	(*TODO: Implement temperature Errors specific to current Cryo MODE (COLD, WARM etc): LOWLOW, LOW, OKAY, HIGH, HIGHHIGH*)
	{attribute 'OPC.UA.DA' := '0'}
	in_lrLowWarning:		LREAL;
	{attribute 'OPC.UA.DA' := '0'}
	in_lrLowLowAlarm:		LREAL;
	{attribute 'OPC.UA.DA' := '0'}
	in_lrHighWarning:		LREAL;
	{attribute 'OPC.UA.DA' := '0'}
	in_HighHighAlarm:		LREAL;
	
END_VAR
VAR
	{attribute 'OPC.UA.DA' := '0'}
	i_fValue	AT%I*:	REAL;    // lower precision, used e.g. by LS240
	{attribute 'OPC.UA.DA' := '0'}
	i_lrValue	AT%I*:  LREAL;   // higher precision, used by other sources
	{attribute 'OPC.UA.DA' := '0'}
    i_bValid    AT%I*:	BOOL;    // valid status, used e.g. by ramp and voters
		
    {attribute 'OPC.UA.DA' := '0'}
	RefStatBase:    REFERENCE TO T_METIS_SENSOR_BASE_STATUS;
	
	{attribute 'OPC.UA.DA' := '0'}
	bRampTimerStarted:	BOOL := FALSE;
	{attribute 'OPC.UA.DA' := '0'}
	rampTimer:	TON;		// Timer for calculating ramp
	
END_VAR

// Set references
RefStat	REF= RefStatBase;


// Get the raw reading and the status of the input channel
M_ReadSensor();

// Calculate value and validity
M_SetStatus();

// Calculate Temperature change ramp
M_GetRamp();

METHOD M_GetRamp
VAR_INPUT
END_VAR
VAR_INST
	{attribute 'OPC.UA.DA' := '0'}
	lrRampStartValueSi: LREAL;	// SI value at start of ramp timer [K]
END_VAR
VAR
	nRampPeriodSec:		UDINT;	// Ramp measurement period [sec].
END_VAR
IF NOT bRampTimerStarted THEN
	bRampTimerStarted	:= TRUE;
	lrRampStartValueSi	:= RefStatBase.lrBaseValue;
	rampTimer(IN:=FALSE);
END_IF

// Execute timer.
// Ramp measurement period should be > 0
nRampPeriodSec	:= in_nRampPeriodSec;
IF nRampPeriodSec = 0 THEN
	nRampPeriodSec	:= 60;
END_IF
rampTimer(IN:=TRUE,PT:=UDINT_TO_TIME(nRampPeriodSec)*1000);

// Calculate ramp at time expiry
IF rampTimer.Q THEN
	// Calculate the temperature ramp per minute
    RefStatBase.lrBaseRamp := (RefStatBase.lrBaseValue - lrRampStartValueSi) * 60.0 / nRampPeriodSec;

	// Current temperature is the starting value of the ramp
	lrRampStartValueSi := RefStatBase.lrBaseValue;

	// Restart the timer
	rampTimer(IN:=FALSE);
END_IF
END_METHOD

// Get input channel status and the raw reading
METHOD M_ReadSensor
VAR_INPUT
END_VAR
VAR_INST
    {attribute 'OPC.UA.DA' := '0'}
    lrPreviousBaseValue : LREAL;
    
    {attribute 'OPC.UA.DA' := '0'}
    _changingValueTimeout : TON;
END_VAR
// Get the base value
CASE in_eSource OF 
    E_METIS_SENSOR_SOURCE.LS240:
        RefStatBase.lrBaseValue := REAL_TO_LREAL(i_fValue) * in_lrScale + in_lrOffset;
    E_METIS_SENSOR_SOURCE.LS336,
    E_METIS_SENSOR_SOURCE.VOTER,
    E_METIS_SENSOR_SOURCE.RAMP,
    E_METIS_SENSOR_SOURCE.DEW_POINT_CALC:
        RefStatBase.lrBaseValue := i_lrValue * in_lrScale + in_lrOffset;
    E_METIS_SENSOR_SOURCE.EL32XX:
        SUPER^.M_ReadSensor();
        RefStatBase.lrBaseValue := INT_TO_LREAL(i_nValue) * in_lrScale + in_lrOffset;
    ELSE
        RefStatBase.lrBaseValue := i_lrValue * in_lrScale + in_lrOffset;
END_CASE

// check if the value is changing
IF RefStatBase.lrBaseValue <> lrPreviousBaseValue THEN
    _changingValueTimeout(IN := FALSE);
    lrPreviousBaseValue := RefStatBase.lrBaseValue;
ELSE
    IF in_eSource = E_METIS_SENSOR_SOURCE.LS240 THEN
        _changingValueTimeout(IN := TRUE, PT := T#20s);
    ELSE
        _changingValueTimeout(IN := TRUE, PT := T#60s);
	END_IF
END_IF

// use the changing value to set the status for sources that don't have a better
// status indication
CASE in_eSource OF 
    E_METIS_SENSOR_SOURCE.EL32XX:
        ; // already set by SUPER^.M_ReadSensor()
    E_METIS_SENSOR_SOURCE.LS240:
        RefStat.bInputUnder	    := FALSE;
        RefStat.bInputOver	    := FALSE;
        RefStat.bInputToggle    := FALSE;
        RefStat.bInputError	    := FALSE;
        RefStat.bInputValid	    := NOT _changingValueTimeout.Q;
        RefStat.bInputActive    := RefStat.bInputValid;
    ELSE
        RefStat.bInputUnder	    := FALSE;
        RefStat.bInputOver	    := FALSE;
        RefStat.bInputToggle    := FALSE;
        RefStat.bInputError	    := NOT i_bValid;
        RefStat.bInputValid     := i_bValid AND (NOT _changingValueTimeout.Q);
        RefStat.bInputActive    := i_bValid AND (NOT _changingValueTimeout.Q);
END_CASE
END_METHOD

METHOD M_SetStatus
VAR_INPUT
END_VAR
// TODO USER: Implement the method.

// copy some input values to the stat object
RefStatBase.eType    := in_eType;
RefStatBase.eSource  := in_eSource;
RefStatBase.sName    := in_sName;

// Update value depending on the sensor type.
// So far, only PT100 supported.

IF RefStat.bInputActive THEN
    
    CASE in_eSource OF
        E_METIS_SENSOR_SOURCE.LS240:
            M_SetStatus_LS240();
        E_METIS_SENSOR_SOURCE.EL32XX:
			RefStat.bError			:= RefStat.bInputError OR RefStat.bInputOver OR RefStat.bInputUnder;
        	RefStat.bValid 	        := NOT RefStat.bError;
        	RefStatBase.bWarning    := FALSE; 
			IF RefStat.bInputOver THEN
        		RefStatBase.sErrorText  := 'OVERRANGE';
			ELSIF RefStat.bInputUnder THEN
        		RefStatBase.sErrorText  := 'UNDERRANGE';
			ELSIF RefStat.bInputError THEN
        		RefStatBase.sErrorText  := 'INPUT ERROR';
			ELSIF RefStat.bError THEN
        		RefStatBase.sErrorText  := 'ERROR';
			ELSE
        		RefStatBase.sErrorText  := 'VALID READING';
			END_IF
    ELSE
        RefStat.bValid 	        := TRUE; 
        RefStat.bError 	        := FALSE;
        RefStatBase.bWarning    := FALSE; 
        RefStatBase.sErrorText  := 'VALID READING';
    END_CASE
ELSE	
	RefStat.bValid	        := FALSE;
	RefStat.bError	        := TRUE;
	RefStatBase.bWarning    := FALSE;
    RefStatBase.sErrorText  := 'INACTIVE';
END_IF
END_METHOD

// Calculate pressure based on the status in input value
METHOD M_SetStatus_LS240
VAR_INPUT
END_VAR
VAR
	lr_MaxRamp:		LREAL := in_lrFaultRamp + 10.0;

	lr_T_LowError:		LREAL := 25.0;
	lr_T_LowWarning:	LREAL := 30.0;
	lr_T_HighWarning:	LREAL := 345.0;
	lr_T_HighError:		LREAL := 346.0;  
END_VAR

IF RefStatBase.lrBaseValue > lr_T_LowWarning AND RefStatBase.lrBaseValue < lr_T_HighWarning AND
    ABS(RefStatBase.lrBaseRamp) < in_lrFaultRamp THEN
    
    RefStat.bValid          := TRUE; 
    RefStatBase.bWarning     := FALSE; 
    RefStat.bError          := FALSE;
    RefStatBase.sErrorText   := 'WITHIN RANGE';
    
ELSIF (RefStatBase.lrBaseValue < lr_T_LowWarning AND RefStatBase.lrBaseValue > lr_T_LowError) OR
        (RefStatBase.lrBaseValue > lr_T_HighWarning AND RefStatBase.lrBaseValue < lr_T_HighError) OR
        ABS(RefStatBase.lrBaseRamp) > in_lrFaultRamp AND ABS(RefStatBase.lrBaseRamp) < lr_MaxRamp THEN

    RefStat.bValid          := TRUE;
    RefStatBase.bWarning     := TRUE;  
    RefStat.bError          := FALSE;
    RefStatBase.sErrorText   := 'WARNING LIMITS EXCEEDED';
    
ELSIF RefStatBase.lrBaseValue < lr_T_LowError OR RefStatBase.lrBaseValue > lr_T_HighError OR
    ABS(RefStatBase.lrBaseRamp) > lr_MaxRamp THEN
    
    RefStat.bValid          := FALSE;
    RefStatBase.bWarning     := FALSE;	   
    RefStat.bError          := TRUE;
    RefStatBase.sErrorText   := 'ERROR LIMITS EXCEEDED';
   
END_IF
END_METHOD

END_FUNCTION_BLOCK

// POUs/Devices/Temp_Sensor/FB_SIM_TEMP_SENSOR_DT670
FUNCTION_BLOCK FB_SIM_TEMP_SENSOR_DT670
VAR_INPUT
	
	//in_lrTempK:		LREAL	:= 100.0;	// Target Temperature [K]
	in_Temp_Sensor_DT670:		FB_METIS_TEMP_SENSOR_DT670;	
	
END_VAR
VAR_OUTPUT
END_VAR
VAR
	sName											: STRING;	

	(* input *)
	bEnable											: BOOL		:= TRUE;
	fStart											: LREAL 	:= 100;
	fTarget											: LREAL		:= 150;
	
	bInit											: BOOL 		:= TRUE; (* To initialize the required ramp*)
	
	(* Ramp *)
	RampUp_Rate										: LREAL		:= 8;	(* in units per Minute *) 
	RampDown_Rate									: LREAL		:= 8;	(* in units per Minute *)
	
	(* function block *)
	fbCTRL_RAMP_GENERATOR							: FB_CTRL_RAMP_GENERATOR;
	stCTRL_RAMP_GENERATOR_PARAMS					: ST_CTRL_RAMP_GENERATOR_PARAMS;	
	
	q_bToggle	AT%Q*:	BOOL	:= FALSE;	// Simulated status
	q_fValue	AT%Q*:	REAL;			// Simulated value [bit]
	
	fOut				: LREAL;		
    bValueReached		: BOOL;
    bError				: BOOL;
    eErrorId			: E_CTRL_ERRORCODES;
	bConfigured			: BOOL;
	
////////////////////////////////////////////////////	
	
	{attribute 'OPC.UA.DA' := '0'}
	toggleTimer:	TON;		// Timer for PDO (alive) toggle
	{attribute 'OPC.UA.DA' := '0'}
	rampTimer:		TON;		// Timer for temperature ramp

	{attribute 'OPC.UA.DA' := '0'}
	nPeriod:		UDINT	:= 10000;	// RAMP/SINE Command period, default 10000ms = 10s
	
	lrTemp_SetPoint:			LREAL;
	
	
END_VAR

// Configuration 

sName := in_Temp_Sensor_DT670.in_sName;

IF bInit THEN
	M_Configure();
END_IF

stCTRL_RAMP_GENERATOR_PARAMS.fVeloPos			:= 0.01666 * RampUp_Rate; (* 1/60 to convert into units per second *)
stCTRL_RAMP_GENERATOR_PARAMS.fVeloNeg			:= 0.01666 * RampDown_Rate; (* 1/60 to convert into units per second *)

//ctrl.fTarget := in_fRampSetPoint;

// Execute Controller
M_ExecuteController();


// lrTempK
q_fValue	:= LREAL_TO_REAL(fOut);

//
// Simulate terminal alive toggle every 160ms.
//
IF NOT bEnable THEN
	bEnable	:= TRUE;
	toggleTimer(IN:=FALSE);
END_IF
toggleTimer(IN:=TRUE,PT:=T#160MS);

q_bToggle	:= toggleTimer.Q;
IF toggleTimer.Q THEN
	q_bToggle	:= toggleTimer.Q;
	toggleTimer(IN:=FALSE);
END_IF

METHOD M_Configure : BOOL
VAR_INPUT
END_VAR


(* init parameter struct *)
	stCTRL_RAMP_GENERATOR_PARAMS.tTaskCycleTime		:= T#10MS;
	stCTRL_RAMP_GENERATOR_PARAMS.tCtrlCycleTime		:= T#10MS;
	stCTRL_RAMP_GENERATOR_PARAMS.fVeloPos			:= 0.01666 * RampUp_Rate; (* 1/60 to convert into units per second *)
	stCTRL_RAMP_GENERATOR_PARAMS.fVeloNeg			:= 0.01666 * RampDown_Rate; (* 1/60 to convert into units per second *)

	(* reset the init flag *)
	bInit							:= FALSE;
END_METHOD

METHOD M_ExecuteController : BOOL
VAR_INPUT
END_VAR
(* call function block *)
fbCTRL_RAMP_GENERATOR(				bEnable					:= bEnable,
									fStart					:= fStart,
									fTarget					:= fTarget,
									stParams				:= stCTRL_RAMP_GENERATOR_PARAMS,
									fOut					=> fOut,
									bValueReached			=> bValueReached,
									bError					=> bError,
									eErrorId				=> eErrorId);
END_METHOD

END_FUNCTION_BLOCK

// POUs/Devices/Temp_Sensor/FB_METIS_TEMP_SENSOR_DT670
FUNCTION_BLOCK FB_METIS_TEMP_SENSOR_DT670
VAR_INPUT
	{attribute 'OPC.UA.DA' := '0'}
	in_sName:				STRING;
	{attribute 'OPC.UA.DA' := '0'}
	in_nLSType:				E_METIS_LAKE_SHORE_TYPE	:= E_METIS_LAKE_SHORE_TYPE.LS240;
	{attribute 'OPC.UA.DA' := '0'}
	in_nRampPeriodSec:		UDINT := 60;		// Ramp measurement period [sec]. Default 60 sec.
	{attribute 'OPC.UA.DA' := '0'}
	in_lrFaultRamp:			LREAL := 10;		// Ramp > in_nFaultRamp OR Ramp < -in_nFaultRamp(deg/min) indicate DT670 sensor fault.	

	(*TODO: Implement temperature Errors specific to current Cryo MODE (COLD, WARM etc): LOWLOW, LOW, OKAY, HIGH, HIGHHIGH*)
	{attribute 'OPC.UA.DA' := '0'}
	in_lrLowWarning:		LREAL;
	{attribute 'OPC.UA.DA' := '0'}
	in_lrLowLowAlarm:		LREAL;
	{attribute 'OPC.UA.DA' := '0'}
	in_lrHighWarning:		LREAL;
	{attribute 'OPC.UA.DA' := '0'}
	in_HighHighAlarm:		LREAL;
	
	in_nCryoMode:			INT; // COLD, COOL_DOWN, WARM_UP, WARM

END_VAR
VAR
//	{attribute 'OPC.UA.DA' := '0'}
//	i_nStatus	AT %I*: UINT;
	{attribute 'OPC.UA.DA' := '0'}
	i_fValue	AT%I*:	REAL;   // lower precision, used by LS240
	{attribute 'OPC.UA.DA' := '0'}
	i_lrValue	AT%I*:  LREAL;   // higher precision, used by other sources
	{attribute 'OPC.UA.DA' := '0'}
	i_bToggle	AT%I*:	BOOL;
	
	{attribute 'OPC.UA.DA' := '0'}
	bStarted:		BOOL := FALSE;
	{attribute 'OPC.UA.DA' := '0'}
	toggleTimer:	TON;		// Timer for PDO (alive) toggle
	{attribute 'OPC.UA.DA' := '0'}
	toggleTrig:		R_TRIG;		// PDO (alive) toggle detection
	
	RefStat: 	REFERENCE TO T_METIS_DT670_TEMP_SENSOR_STATUS;
	
	{attribute 'OPC.UA.DA' := '0'}
	stat:	T_METIS_DT670_TEMP_SENSOR_STATUS;	// Complete status

	{attribute 'OPC.UA.DA' := '0'}
	bRampTimerStarted:	BOOL := FALSE;
	{attribute 'OPC.UA.DA' := '0'}
	rampTimer:	TON;		// Timer for calculating ramp
	
END_VAR

// Set references
RefStat	REF=stat;


// Get the raw reading and the status of the input channel
M_ReadSensor();

// Calculate value and validity
M_SetStatus();

// Calculate Temperature change ramp
M_GetRamp();

METHOD M_GetRamp
VAR_INPUT
END_VAR
VAR_INST
	{attribute 'OPC.UA.DA' := '0'}
	lrRampStartTempK:	LREAL;	// Temperature at start of ramp timer [K]
END_VAR
VAR
	nRampPeriodSec:		UDINT;	// Ramp measurement period [sec].
END_VAR
IF NOT bRampTimerStarted THEN
	bRampTimerStarted	:= TRUE;
	lrRampStartTempK	:= stat.lrTempK;
	rampTimer(IN:=FALSE);
END_IF

// Execute timer.
// Ramp measurement period should be > 0
nRampPeriodSec	:= in_nRampPeriodSec;
IF nRampPeriodSec = 0 THEN
	nRampPeriodSec	:= 60;
END_IF
rampTimer(IN:=TRUE,PT:=UDINT_TO_TIME(nRampPeriodSec)*1000);

// Calculate ramp at time expiry
IF rampTimer.Q THEN
	// Calculate the temperature ramp per minute
//	IF stat.bValid THEN
		stat.lrRamp	:= (stat.lrTempK - lrRampStartTempK) * 60.0 / nRampPeriodSec;
//	ELSE
//		stat.lrRamp	:= 0.0;
//	END_IF

	// Current temperature is the starting value of the ramp
	lrRampStartTempK	:= stat.lrTempK;

	// Restart the timer
	rampTimer(IN:=FALSE);
END_IF
END_METHOD

// Get input channel status and the raw reading
METHOD M_ReadSensor
VAR_INPUT
END_VAR
VAR_INST
    fPreviousValue : REAL;
END_VAR
// Get input channel status
//RefStat.bInputUnder	:= (i_nStatus AND 2#0000_0000_0000_0001) <> 0;
//RefStat.bInputOver	:= (i_nStatus AND 2#0000_0000_0000_0010) <> 0;
//RefStat.bInputError	:= (i_nStatus AND 2#0000_0000_0100_0000) <> 0;
//RefStat.bInputToggle:= (i_nStatus AND 2#1000_0000_0000_0000) <> 0;
//RefStat.bInputValid	:= (i_nStatus AND 2#0100_0000_0000_0000)  = 0;	// 0 -> PDO OK

// Get the raw reading
CASE in_nLSType OF 
    E_METIS_LAKE_SHORE_TYPE.LS240:
        RefStat.lrRawValue	:= REAL_TO_LREAL(i_fValue);
    E_METIS_LAKE_SHORE_TYPE.LS336,
    E_METIS_LAKE_SHORE_TYPE.VOTER,
    E_METIS_LAKE_SHORE_TYPE.RAMP:
        RefStat.lrRawValue	:= i_lrValue;
        RefStat.lrRawValue	:= i_lrValue;
    ELSE
        RefStat.lrRawValue	:= i_lrValue;
END_CASE

// for LS240, we don't have an explicit toggle flag.
// But in reality the raw value is continuously changing (due to noise)
// so we use a change of the raw value as a toggle
IF fPreviousValue <> i_fValue AND in_nLSType = E_METIS_LAKE_SHORE_TYPE.LS240 THEN
    i_bToggle := NOT i_bToggle;
    fPreviousValue := i_fValue;
END_IF

RefStat.bInputToggle:= i_bToggle;

//
// Check if the terminal is alive.
// Start the time that will expire in 3 sec.
// If bToggle bit triggers before the timer expires, 
// this is the sign that the terminal is alive.
//
IF NOT bStarted THEN
	bStarted	:= TRUE;
	toggleTimer(IN:=FALSE);
END_IF
toggleTimer(IN:=TRUE,PT:=T#3S);
toggleTrig(CLK:=RefStat.bInputToggle);

IF toggleTrig.Q THEN
	// bToggle bit has triggered. Terminal is alive.
	RefStat.bInputActive	:= TRUE;
	// Restart the timer
	toggleTimer(IN:=FALSE);
ELSIF toggleTimer.Q THEN
	// bInputToggle bit has not triggered within 3 sec. Terminal is NOT alive.
	RefStat.bInputActive	:= FALSE;
	// Restart the timer
	toggleTimer(IN:=FALSE);
END_IF
END_METHOD

// Calculate pressure based on the status in input value
METHOD M_SetSensorStatus_DT670_LS240
VAR_INPUT
END_VAR
VAR
	lr_MaxRamp:		LREAL := in_lrFaultRamp + 5.0;

	lr_T_LowError:		LREAL := 25.0;
	lr_T_LowWarning:	LREAL := 30.0;
	lr_T_HighWarning:	LREAL := 300.0;
	lr_T_HighError:		LREAL := 345.0;  
END_VAR
//
// Set the temperature as it is read.
// Later on we decide if it is valid or not.
//

stat.lrTempK 	:= stat.lrRawValue;		// Raw value is recorderd as Kelvin
stat.lrTempC 	:= stat.lrTempK - 273.15; 

//
// Update validity

IF stat.bInputActive THEN
	
    IF stat.lrTempK > lr_T_LowWarning AND stat.lrTempK < lr_T_HighWarning AND
		ABS(stat.lrRamp) < in_lrFaultRamp THEN
		
		stat.bValid 	:= 		TRUE; 
		stat.bWarning 	:= 		FALSE; 
		stat.bError 	:= 		FALSE;
        stat.sErrorText :=      'WITHIN RANGE';
		
	ELSIF (stat.lrTempK < lr_T_LowWarning AND stat.lrTempK > lr_T_LowError) OR
			(stat.lrTempK > lr_T_HighWarning AND stat.lrTempK < lr_T_HighError) OR
			ABS(stat.lrRamp) > in_lrFaultRamp AND ABS(stat.lrRamp) < lr_MaxRamp THEN
		stat.bValid 	:= 		TRUE;
		stat.bWarning 	:= 		TRUE;  
		stat.bError 	:= 		FALSE;
        stat.sErrorText :=      'WARNING LIMITS EXCEEDED';
		
	ELSIF stat.lrTempK < lr_T_LowError OR stat.lrTempK > lr_T_HighError OR
		ABS(stat.lrRamp) > lr_MaxRamp THEN
		
	   	stat.bValid 	:= 		FALSE;
		stat.bWarning 	:= 		FALSE;	   
		stat.bError 	:= 		TRUE;
        stat.sErrorText :=      'ERROR LIMITS EXCEEDED';
	   
	END_IF



//	IF ABS(stat.lrRamp) < in_lrFaultRamp THEN
//					stat.bValid 	:= 		TRUE; 
//					stat.bWarning 	:= 		FALSE; 
//					stat.bError 	:= 		FALSE;
//	ELSIF ABS(stat.lrRamp) > in_lrFaultRamp AND ABS(stat.lrRamp) < lr_MaxRamp THEN
//					stat.bValid 	:= 		TRUE; 
//					stat.bWarning 	:= 		TRUE; 
//					stat.bError 	:= 		FALSE;
//	ELSIF ABS(stat.lrRamp) > lr_MaxRamp THEN
//					stat.bValid 	:= 		FALSE; 
//					stat.bWarning 	:= 		FALSE; 
//					stat.bError 	:= 		TRUE;
//	END_IF



		
ELSE	
	stat.bValid	:= FALSE;
	stat.bWarning := FALSE;
	stat.bError	:= TRUE;
    stat.sErrorText := 'INACTIVE';
END_IF	

	//	IF stat.lrRamp < in_lrFaultRamp THEN
//					stat.bValid 	:= 		TRUE; 
//					stat.bWarning 	:= 		FALSE; 
//					stat.bError 	:= 		FALSE;
//	ELSIF stat.lrRamp > in_lrFaultRamp AND stat.lrRamp < lr_MaxRamp THEN
//					stat.bValid 	:= 		TRUE; 
//					stat.bWarning 	:= 		TRUE; 
//					stat.bError 	:= 		FALSE;
//	ELSIF stat.lrRamp > lr_MaxRamp THEN
//					stat.bValid 	:= 		FALSE; 
//					stat.bWarning 	:= 		FALSE; 
//					stat.bError 	:= 		TRUE;
//	END_IF
END_METHOD

// Calculate pressure based on the status in input value
METHOD M_SetSensorStatus_DT670_LS336
VAR_INPUT
END_VAR
VAR
END_VAR

stat.lrTempK 	:= stat.lrRawValue;		// Raw value is recorderd as Kelvin
stat.lrTempC 	:= stat.lrTempK - 273.15; 

//
// Update validity

IF stat.bInputActive THEN
    stat.bValid 	:= TRUE; 
    stat.bWarning 	:= FALSE; 
    stat.bError 	:= FALSE;
    stat.sErrorText := 'VALID READING';
ELSE	
	stat.bValid	    := FALSE;
	stat.bWarning   := FALSE;
	stat.bError	    := TRUE;
    stat.sErrorText := 'INACTIVE';
END_IF
END_METHOD

METHOD M_SetSensorStatus_DT670_Ramp
VAR_INPUT
END_VAR

stat.lrTempK 	:= stat.lrRawValue;		// Raw value is recorderd as Kelvin
stat.lrTempC 	:= stat.lrTempK - 273.15; 

//
// Update validity

IF stat.bInputActive THEN
    stat.bValid 	:= TRUE; 
    stat.bWarning 	:= FALSE; 
    stat.bError 	:= FALSE;
    stat.sErrorText := 'VALID READING';
ELSE	
	stat.bValid	    := FALSE;
	stat.bWarning   := FALSE;
	stat.bError	    := TRUE;
    stat.sErrorText := 'INACTIVE';
END_IF
END_METHOD

METHOD M_SetSensorStatus_DT670_Voter
VAR_INPUT
END_VAR

stat.lrTempK 	:= stat.lrRawValue;		// Raw value is recorderd as Kelvin
stat.lrTempC 	:= stat.lrTempK - 273.15; 

//
// Update validity

IF stat.bInputActive THEN
    stat.bValid 	:= TRUE; 
    stat.bWarning 	:= FALSE; 
    stat.bError 	:= FALSE;
    stat.sErrorText := 'VALID READING';
ELSE	
	stat.bValid	    := FALSE;
	stat.bWarning   := FALSE;
	stat.bError	    := TRUE;
    stat.sErrorText := 'INACTIVE';
END_IF
END_METHOD

METHOD M_SetStatus
VAR_INPUT
END_VAR
// TODO USER: Implement the method.

// Set LakeShore type
stat.nLSType	:= in_nLSType;
stat.sName		:= in_sName;
// Update value depending on the sensor type.
// So far, only PT100 supported.
CASE in_nLSType OF
	E_METIS_LAKE_SHORE_TYPE.LS240:
		M_SetSensorStatus_DT670_LS240();
	E_METIS_LAKE_SHORE_TYPE.LS336:
		M_SetSensorStatus_DT670_LS336();
	E_METIS_LAKE_SHORE_TYPE.VOTER:
        M_SetSensorStatus_DT670_Voter();
	E_METIS_LAKE_SHORE_TYPE.RAMP:
        M_SetSensorStatus_DT670_Ramp();
END_CASE

(*

TODO Implement

in_lrLowWarning:		LREAL;	
in_lrLowLowAlarm:		LREAL;
in_lrHighWarning:		LREAL;
in_HighHighAlarm:		LREAL;
	
bLowWarning:
bLowLowAlarm:	
bHighWarning:	
bHighHighAlarm:	

stat.sErrorText :=  'Low Warning'
stat.sErrorText := 	'Low Low Alarm'	
stat.sErrorText :=	'High Warning'	
stat.sErrorText :=	'High High Alarm'	


*)
END_METHOD

METHOD M_SetTemperature : LREAL
VAR_INPUT
END_VAR
M_SetTemperature := stat.lrTempK;
END_METHOD

END_FUNCTION_BLOCK

// POUs/Devices/Heaters/FB_METIS_HEATERS
FUNCTION_BLOCK FB_METIS_HEATERS
VAR_INPUT
END_VAR
VAR_OUTPUT
END_VAR
VAR_IN_OUT
	{attribute 'OPC.UA.DA' := '0'}
    tctrl:                  FB_METIS_TCTRL;
END_VAR
VAR
	{attribute 'TcHmiSymbol.Show'}
    h_cry_sha:              FB_METIS_HEATER;
	{attribute 'TcHmiSymbol.Show'}
    h_cry_shb:              FB_METIS_HEATER;
	{attribute 'TcHmiSymbol.Show'}
    h_cry_shc:              FB_METIS_HEATER;
	{attribute 'TcHmiSymbol.Show'}
    h_cry_sp:               FB_METIS_HEATER;    
    h_cry_pta:              FB_METIS_HEATER;   // PTC A (LMS) Ear Flange        H_CRY_PTA
    h_cry_ptb:              FB_METIS_HEATER;   // PTC B (IMG) Ear Flange        H_CRY_PTB
    h_cry_ptc:              FB_METIS_HEATER;   // PTC C (IMG DETs) Ear Flange   H_CRY_PTC
    h_cry_wi:               FB_METIS_HEATER;   // Window heater (PWM)
    
    h_img_wuh_1:            FB_METIS_HEATER;   // IMG WUH circuit 1
    h_img_wuh_2:            FB_METIS_HEATER;   // IMG WUH circuit 2
    h_img_lmd_2:            FB_METIS_HEATER;   // IMG LM-band detector heater SPARE
    h_img_lmp_2:            FB_METIS_HEATER;   // IMG LM-band preamp heater SPARE
    h_img_nd_2:             FB_METIS_HEATER;   // IMG N-band detector heater SPARE
    
    h_sca_wuh_1:            FB_METIS_HEATER;   // SCA WUH circuit 1
    h_sca_wuh_2:            FB_METIS_HEATER;   // SCA WUH circuit 2
    h_sca_det_2:            FB_METIS_HEATER;   // SCA detector heater SPARE
    h_sca_dhs_2:            FB_METIS_HEATER;   // IMG detector heat sink heater SPARE
END_VAR

M_ExecuteControllers(tctrl);

METHOD M_ExecuteControllers
VAR_INPUT
END_VAR
VAR_IN_OUT
    tctrl: FB_METIS_TCTRL;
END_VAR
h_cry_sha(
    in_sName                := 'H_CRY_SHA',
    in_lrHeaterResistance   := 10,
    in_lrHeaterMaxPower     := 360,
    in_eHeaterType          := E_METIS_CRYO_HEATER_TYPE.CPAU60,
    in_sAutoSetpointSource  := tctrl.tc_cry_sha.in_sName,
    in_lrAutoSetpointValue  := tctrl.tc_cry_sha.stat.lrControllerOut);
h_cry_shb(
    in_sName                := 'H_CRY_SHB',
    in_lrHeaterResistance   := 10,
    in_lrHeaterMaxPower     := 360,
    in_eHeaterType          := E_METIS_CRYO_HEATER_TYPE.CPAU60,
    in_sAutoSetpointSource  := tctrl.tc_cry_shb.in_sName,
    in_lrAutoSetpointValue  := tctrl.tc_cry_shb.stat.lrControllerOut);
h_cry_shc(
    in_sName                := 'H_CRY_SHC',
    in_lrHeaterResistance   := 10,
    in_lrHeaterMaxPower     := 360,
    in_eHeaterType          := E_METIS_CRYO_HEATER_TYPE.CPAU60,
    in_sAutoSetpointSource  := tctrl.tc_cry_shc.in_sName,
    in_lrAutoSetpointValue  := tctrl.tc_cry_shc.stat.lrControllerOut);
h_cry_sp(
    in_sName                := 'H_CRY_SP',
    in_lrHeaterResistance   := 12.5,
    in_lrHeaterMaxPower     := 42,
    in_eHeaterType          := E_METIS_CRYO_HEATER_TYPE.PWM_SORPTION,
	in_lrAutoSetpointValue  := tctrl.tc_cry_sp.stat.lrControllerOut);
	
h_cry_pta(
    in_sName                := 'H_CRY_PTA',
    in_lrHeaterResistance   := 40,
    in_lrHeaterMaxPower     := 90,
    in_eHeaterType          := E_METIS_CRYO_HEATER_TYPE.CXWUI60,
    in_sAutoSetpointSource  := tctrl.tc_cry_pt.in_sName,
    in_lrAutoSetpointValue  := tctrl.tc_cry_pt.stat.lrControllerOut);
h_cry_ptb(
    in_sName                := 'H_CRY_PTB',
    in_lrHeaterResistance   := 40,
    in_lrHeaterMaxPower     := 90,
    in_eHeaterType          := E_METIS_CRYO_HEATER_TYPE.CXWUI60,
    in_sAutoSetpointSource  := tctrl.tc_cry_pt.in_sName,
    in_lrAutoSetpointValue  := tctrl.tc_cry_pt.stat.lrControllerOut);
h_cry_ptc(
    in_sName                := 'H_CRY_PTC',
    in_lrHeaterResistance   := 40,
    in_lrHeaterMaxPower     := 90,
    in_eHeaterType          := E_METIS_CRYO_HEATER_TYPE.CXWUI60,
    in_sAutoSetpointSource  := tctrl.tc_cry_pt.in_sName,
    in_lrAutoSetpointValue  := tctrl.tc_cry_pt.stat.lrControllerOut);
h_cry_wi(
    in_sName                := 'H_CRY_WI',
    in_lrHeaterResistance   := 12.5,
    in_lrHeaterMaxPower     := 46,
    in_eHeaterType          := E_METIS_CRYO_HEATER_TYPE.PWM_WINDOW,
    in_sAutoSetpointSource  := tctrl.tc_cry_wi.in_sName,
    in_lrAutoSetpointValue  := tctrl.tc_cry_wi.stat.lrControllerOut);

// IMG
h_img_wuh_1(
    in_sName                := 'H_IMG_WUH_1', 
    in_lrHeaterResistance   := 10, 
    in_lrHeaterMaxPower     := 360, 
    in_eHeaterType          := E_METIS_CRYO_HEATER_TYPE.CPAU60,
    in_sAutoSetpointSource  := tctrl.tc_img_wuh.in_sName,
    in_lrAutoSetpointValue  := tctrl.tc_img_wuh.stat.lrControllerOut);
h_img_wuh_2(
    in_sName                := 'H_IMG_WUH_2',
    in_lrHeaterResistance   := 10,
    in_lrHeaterMaxPower     := 360,
    in_eHeaterType          := E_METIS_CRYO_HEATER_TYPE.CPAU60,
    in_sAutoSetpointSource  := tctrl.tc_img_wuh.in_sName,
    in_lrAutoSetpointValue  := tctrl.tc_img_wuh.stat.lrControllerOut);
h_img_lmd_2(
    in_sName                := 'H_IMG_LMD_2',
    in_lrHeaterResistance   := 75,
    in_lrHeaterMaxPower     := 5,
    in_eHeaterType          := E_METIS_CRYO_HEATER_TYPE.PWM_DETECTOR,
    in_sAutoSetpointSource  := tctrl.tc_img_lmd_2.in_sName,
    in_lrAutoSetpointValue  := tctrl.tc_img_lmd_2.stat.lrControllerOut);
h_img_lmp_2(
    in_sName                := 'H_IMG_LMP_2',
    in_lrHeaterResistance   := 24,
    in_lrHeaterMaxPower     := 5,
    in_eHeaterType          := E_METIS_CRYO_HEATER_TYPE.PWM_DETECTOR,
    in_sAutoSetpointSource  := tctrl.tc_img_lmp_2.in_sName,
    in_lrAutoSetpointValue  := tctrl.tc_img_lmp_2.stat.lrControllerOut);
h_img_nd_2(
    in_sName                := 'H_IMG_ND_2',
    in_lrHeaterResistance   := 75,
    in_lrHeaterMaxPower     := 5,
    in_eHeaterType          := E_METIS_CRYO_HEATER_TYPE.PWM_DETECTOR,
    in_sAutoSetpointSource  := tctrl.tc_img_nd_2.in_sName,
    in_lrAutoSetpointValue  := tctrl.tc_img_nd_2.stat.lrControllerOut);

// SCA
h_sca_wuh_1(
    in_sName                := 'H_SCA_WUH_1', 
    in_lrHeaterResistance   := 10,
    in_lrHeaterMaxPower     := 360,
    in_eHeaterType          := E_METIS_CRYO_HEATER_TYPE.CPAU60,
    in_sAutoSetpointSource  := tctrl.tc_sca_wuh.in_sName,
    in_lrAutoSetpointValue  := tctrl.tc_sca_wuh.stat.lrControllerOut);
h_sca_wuh_2(
    in_sName                := 'H_SCA_WUH_2',
    in_lrHeaterResistance   := 10,
    in_lrHeaterMaxPower     := 360,
    in_eHeaterType          := E_METIS_CRYO_HEATER_TYPE.CPAU60,
    in_sAutoSetpointSource  := tctrl.tc_sca_wuh.in_sName,
    in_lrAutoSetpointValue  := tctrl.tc_sca_wuh.stat.lrControllerOut);
h_sca_det_2(
    in_sName                := 'H_SCA_DET_2',
    in_lrHeaterResistance   := 75,
    in_lrHeaterMaxPower     := 5,
    in_eHeaterType          := E_METIS_CRYO_HEATER_TYPE.EL95X1,
    in_sAutoSetpointSource  := tctrl.tc_sca_det_2.in_sName,
    in_lrAutoSetpointValue  := tctrl.tc_sca_det_2.stat.lrControllerOut);
h_sca_dhs_2(
    in_sName                := 'H_SCA_DHS_2',
    in_lrHeaterResistance   := 75,
    in_lrHeaterMaxPower     := 5,
    in_eHeaterType          := E_METIS_CRYO_HEATER_TYPE.EL95X1,
    in_sAutoSetpointSource  := tctrl.tc_sca_dhs_2.in_sName,
    in_lrAutoSetpointValue  := tctrl.tc_sca_dhs_2.stat.lrControllerOut);
END_METHOD

END_FUNCTION_BLOCK

// POUs/Control/TCtrl/FB_METIS_TCTRL
FUNCTION_BLOCK FB_METIS_TCTRL
VAR_INPUT
END_VAR
VAR_OUTPUT
END_VAR
VAR_IN_OUT
	{attribute 'OPC.UA.DA' := '0'}
    temperatures:   FB_METIS_TEMPERATURES;  // all temperatures
END_VAR
VAR
    // CRY
	{attribute 'TcHmiSymbol.Show'}
    tc_cry_sha:     FB_METIS_CTRL_TEMPERATURE; // Shield A
    tc_cry_shb:     FB_METIS_CTRL_TEMPERATURE; // Shield B
    tc_cry_shc:     FB_METIS_CTRL_TEMPERATURE; // Shield C
    tc_cry_pt:      FB_METIS_CTRL_TEMPERATURE; // PTC A/B/C
    tc_cry_wi:      FB_METIS_CTRL_TEMPERATURE; // Window
	tc_cry_sp:      FB_METIS_CTRL_TEMPERATURE; // Sorption Pump

    // IMG
    tc_img_wuh:	    FB_METIS_CTRL_TEMPERATURE; // IMG WUH circuits (1 and 2)
    tc_img_lmd_2:	FB_METIS_CTRL_TEMPERATURE; // IMG LM-band detector heater SPARE
    tc_img_lmp_2:	FB_METIS_CTRL_TEMPERATURE; // IMG LM-band preamp heater SPARE
    tc_img_nd_2:	FB_METIS_CTRL_TEMPERATURE; // IMG N-band detector heater SPARE
    
    // SCA
    tc_sca_wuh:	    FB_METIS_CTRL_TEMPERATURE; // SCA WUH circuits (1 and 2)
    tc_sca_det_2:   FB_METIS_CTRL_TEMPERATURE; // SCA detector heater SPARE control
    tc_sca_dhs_2:   FB_METIS_CTRL_TEMPERATURE; // IMG detector heat sink heater SPARE control
END_VAR
VAR CONSTANT
	{attribute 'OPC.UA.DA' := '0'}
    CYCLE_TIME : TIME := T#10ms;
END_VAR

// CRY
tc_cry_sha(in_sName := 'TC_CRY_SHA' , in_tCycleTime := CYCLE_TIME, temperatures := temperatures);
tc_cry_shb(in_sName := 'TC_CRY_SHB' , in_tCycleTime := CYCLE_TIME, temperatures := temperatures);
tc_cry_shc(in_sName := 'TC_CRY_SHC' , in_tCycleTime := CYCLE_TIME, temperatures := temperatures);
tc_cry_pt( in_sName := 'TC_CRY_PT' , in_tCycleTime := CYCLE_TIME, temperatures := temperatures);
tc_cry_wi( in_sName := 'TC_CRY_WI'  , in_tCycleTime := CYCLE_TIME, temperatures := temperatures);
tc_cry_sp( in_sName := 'TC_CRY_SP'  , in_tCycleTime := CYCLE_TIME, temperatures := temperatures);

// IMG
tc_img_wuh(in_sName   := 'TC_IMG_WUH'   , in_tCycleTime := CYCLE_TIME, temperatures := temperatures);
tc_img_lmd_2(in_sName := 'TC_IMG_LMD_2' , in_tCycleTime := CYCLE_TIME, temperatures := temperatures);
tc_img_lmp_2(in_sName := 'TC_IMG_LMP_2' , in_tCycleTime := CYCLE_TIME, temperatures := temperatures);
tc_img_nd_2(in_sName  := 'TC_IMG_ND_2'  , in_tCycleTime := CYCLE_TIME, temperatures := temperatures);

// SCA
tc_sca_wuh(in_sName   := 'TC_SCA_WUH'   , in_tCycleTime := CYCLE_TIME, temperatures := temperatures);
tc_sca_det_2(in_sName := 'TC_SCA_DET_2' , in_tCycleTime := CYCLE_TIME, temperatures := temperatures);
tc_sca_dhs_2(in_sName := 'TC_SCA_DHS_2' , in_tCycleTime := CYCLE_TIME, temperatures := temperatures);

END_FUNCTION_BLOCK

// POUs/Control/Control/FB_METIS_CTRL_TEMPERATURE
FUNCTION_BLOCK FB_METIS_CTRL_TEMPERATURE
VAR_INPUT
	{attribute 'OPC.UA.DA' := '0'}
	in_sName : STRING;   // name of the controller
	{attribute 'OPC.UA.DA' := '0'}
    in_tCycleTime : TIME := T#10ms;
END_VAR
VAR_IN_OUT
	{attribute 'OPC.UA.DA' := '0'}
    temperatures : FB_METIS_TEMPERATURES;  // all temperatures
END_VAR
VAR_OUTPUT
END_VAR
VAR
    // configuration
	{attribute 'OPC.UA.DA' := '0'}
	{attribute 'TcHmiSymbol.Show'}
	fbTcConfig : FB_READ_WRITE_METIS_CTRL_DT670_CFG;
    
    // standard objects
	{attribute 'TcHmiSymbol.Show'}
    stat : T_METIS_CTRL_LOOP_STAT;
	{attribute 'TcHmiSymbol.Show'}
    ctrl : T_METIS_CTRL_LOOP_CTRL;
	{attribute 'TcHmiSymbol.Show'}
    cfg  : T_METIS_CTRL_LOOP_CFG;
    
    
	{attribute 'OPC.UA.DA' := '0'}
		{attribute 'TcHmiSymbol.Show'}
    pInputTemp : POINTER TO FB_METIS_TEMPERATURE;
	{attribute 'OPC.UA.DA' := '0'}
		{attribute 'TcHmiSymbol.Show'}
    pSetpointTemp : POINTER TO FB_METIS_TEMPERATURE;
    
    // Beckhoff controller
	{attribute 'OPC.UA.DA' := '0'}
		{attribute 'TcHmiSymbol.Show'}
	fbCtrlPid       : FB_CTRL_PID;
	{attribute 'OPC.UA.DA' := '0'}
		{attribute 'TcHmiSymbol.Show'}
	stCtrlPidParams : ST_CTRL_PID_PARAMS;
    
	// ramp generator
	ramp: FB_METIS_CTRL_RAMP_GENERATOR;
    
    // array for setpoint selection, used by the HMI
	{attribute 'OPC.UA.DA' := '0'}
		{attribute 'TcHmiSymbol.Show'}
    aSetpointSwitchNames : ARRAY[0..1] OF STRING := [ 'Fixed', 'Variable' ]; 
	
	
				// Alarm handling
	// List of alarms to be handled by Temperature
	arrEventEntry : ARRAY [0..4] OF TcEventEntry;
	// Alarm handler FB
	fbAlarmHandler : FB_AlarmHandler;
	{attribute 'TcHmiSymbol.Show'}
	{attribute 'TcHmiSymbol.ReadOnly'}
	sInstanceName : T_MaxString;
	{attribute 'TcHmiSymbol.Show'}
	bConfirmAllAlarms : BOOL;
	{attribute 'TcHmiSymbol.Show'}
	{attribute 'TcHmiSymbol.ReadOnly'}
	sEventClassName : T_MaxString;
	
	// Logs logs
	logs:	FB_CRYO_FUNCTION_LOG;
    
END_VAR

// to avoid any problem of invalid pointers, set them right away
M_UpdateTempPointers(temperatures := temperatures);

// Read/write configuration
fbTcConfig(in_sTempCtrlName:= in_sName, Temp_Ctrl_Config:= cfg);

// configure during the first cycles
IF NOT stat.bConfigured THEN
    M_Configure(temperatures := temperatures);
    RETURN;
END_IF

// read/write the config (if needed)
M_Read_Write_Config(temperatures := temperatures);


IF stat.bStarted THEN
    M_ExecuteModes();
    M_ExecuteController();
ELSE
    M_Startup();
END_IF

M_UpdateStatus();

IF ctrl.bClearForcedManualDiag THEN
    stat.sLastForcedManualTime := '';
    stat.sLastForcedManualCause := '';
    ctrl.bClearForcedManualDiag := FALSE;
END_IF

// Handle alarms
M_UpdateAlarms();


// Setting Power to the heater
//IF bEngMode AND (NOT ctrl.bEnable) THEN
//	lrControllerOut := lrManualOut; // set manual power
//ELSE
//	lrManualOut := lrControllerOut; // Bumpless transition
//END_IF

METHOD M_ConfigReadingFinished
VAR_INPUT
    bError : BOOL;
END_VAR
VAR_IN_OUT
    temperatures : FB_METIS_TEMPERATURES;
END_VAR
VAR
    i : INT;
END_VAR
IF bError THEN
    // ERROR! Just put the indexes to 0
    ctrl.nInputTempIndex    := 0;
    ctrl.nSetpointTempIndex := 0;
    //ctrl.lrOutMaxLimit              := 100.0;    // TODO
    //ctrl.lrOutMinLimit              := 0.0;      // TODO

ELSE
    // success!
    // update some level-based ctrl variables
    ctrl.nInputTempIndex     := temperatures.M_GetTempSensorIndex(cfg.sInputTempName);
    ctrl.nSetpointTempIndex  := temperatures.M_GetTempSensorIndex(cfg.sSetpointTempName);
    ctrl.lrFixedSetpoint     := cfg.lrFixedSetpoint;
    ctrl.lrSetpointOffset    := cfg.lrSetpointOffset;
    ctrl.lrManualOut         := cfg.lrManualOut;
    // edge-based ctrl variables are better directly updated in stat
    stat.eCtrlMode           := cfg.eStartupCtrlMode;
    //ctrl.lrOutMaxLimit := cfg.lrOutMaxLimit;    // TODO
    //ctrl.lrOutMinLimit := cfg.lrOutMinLimit;    // TODO
END_IF

M_UpdateTempPointers(temperatures := temperatures);

// clear the flag
fbTcConfig.M_ClearReadingDoneFlag();
END_METHOD

METHOD M_Configure : BOOL
VAR_INST
	{attribute 'OPC.UA.DA' := '0'}
    nConfigureState : INT;
END_VAR
VAR_IN_OUT
	{attribute 'OPC.UA.DA' := '0'}
    temperatures : FB_METIS_TEMPERATURES;
END_VAR
VAR
    i : INT;
END_VAR
arrEventEntry[0] := Tc_Events.METISCryoPIDCtrlEventClass.InputTemperatureInvalid;
arrEventEntry[1] := Tc_Events.METISCryoPIDCtrlEventClass.VariableSetpointInvalid;
arrEventEntry[2] := Tc_Events.METISCryoPIDCtrlEventClass.ControllerForcedManual;
arrEventEntry[3] := Tc_Events.METISCryoPIDCtrlEventClass.PidBlockError;
arrEventEntry[4] := Tc_Events.METISCryoPIDCtrlEventClass.RampBlockError;


CASE nConfigureState OF
    0:  
        // configure the base PID controller
        // init parameter struct
        stCtrlPidParams.tCtrlCycleTime	:= in_tCycleTime;
        stCtrlPidParams.tTaskCycleTime	:= in_tCycleTime;
        stCtrlPidParams.fOutMaxLimit    := 100.0;
        stCtrlPidParams.fOutMinLimit    := 0.0;
        // use the name of the control loop as the default description
        cfg.sDescription                := in_sName;
        // ensure some more default settings
        cfg.bEnabled                    := FALSE;
        stat.eCtrlMode                  := E_METIS_CTRL_MODE.MANUAL; 
        // start reading the config
        fbTcConfig.M_ReadConfiguration();
        nConfigureState := 1;
    1:
        IF fbTcConfig.bReadingDoneFlag THEN
            M_ConfigReadingFinished(
                bError       := fbTcConfig.bReadError,
                temperatures := temperatures);
            
            stat.bConfigured := TRUE;
        END_IF
END_CASE
END_METHOD

METHOD M_ExecuteController
VAR_INPUT
END_VAR
VAR_INST
	{attribute 'OPC.UA.DA' := '0'}
	eCtrlMode       : E_CTRL_MODE;
    
	{attribute 'OPC.UA.DA' := '0'}
    bEnableRamp : BOOL;
    
	{attribute 'OPC.UA.DA' := '0'}
    lrActualValue : LREAL;
END_VAR

// set the raw control mode
IF NOT cfg.bEnabled THEN
    stat.lrControllerOut := 0.0;
    stat.bError := FALSE;
    stat.bWarning := FALSE;
    stat.bValid := FALSE;
    RETURN;

ELSIF stat.eCtrlMode = E_METIS_CTRL_MODE.MANUAL THEN
    eCtrlMode := E_CTRL_MODE.eCTRL_MODE_MANUAL;
    // ramp generator should not be running
    bEnableRamp := FALSE;
ELSE
    eCtrlMode := E_CTRL_MODE.eCTRL_MODE_ACTIVE;
    // ramp generator should be running
    bEnableRamp := TRUE;
END_IF

// update the internal control params
stCtrlPidParams.fKp := cfg.lrKp;
stCtrlPidParams.tTn := LREAL_TO_TIME(cfg.lrTn * 1000.0);
stCtrlPidParams.tTd := LREAL_TO_TIME(cfg.lrTd * 1000.0);
stCtrlPidParams.tTv := LREAL_TO_TIME(cfg.lrTv * 1000.0);

// update more stat values
IF ctrl.nSetpointTempIndex <> 0 THEN
    stat.lrActVariableSetpoint := pSetpointTemp^.stat.lrTempK;
ELSE
    stat.lrActVariableSetpoint := 0.0;
END_IF

// calculate the input for the ramp
IF cfg.eSetpointSwitch = E_METIS_CTRL_SETPOINT_SWITCH.FIXED THEN
    stat.lrTargetSetpoint := ctrl.lrFixedSetpoint + ctrl.lrSetpointOffset;
ELSE 
    stat.lrTargetSetpoint := stat.lrActVariableSetpoint + ctrl.lrSetpointOffset;
END_IF

// update the input
stat.lrActInput := pInputTemp^.stat.lrTempK;

// execute the ramp
ramp(
    in_bEnable          := bEnableRamp,
	in_fRampSetPoint	:= stat.lrTargetSetpoint,
    in_fStartPoint      := stat.lrActInput,
 	in_fRampUp_Rate	    := cfg.lrRampUpRate,
 	in_fRampDown_Rate   := cfg.lrRampDownRate,
 	out_fRampValue      => stat.lrRampValue);

// execute the PID algorithm
fbCtrlPid(
    fSetpointValue  := stat.lrRampValue,
    fActualValue    := stat.lrActInput,
    fManSyncValue   := ctrl.lrManualOut,
    bSync           := FALSE,
    eMode           := eCtrlMode,
    bHold           := ctrl.bHold,
    stParams        := stCtrlPidParams,
    fOut            => stat.lrControllerOut,
    bARWactive      => stat.bARWactive,
    bError          => stat.bError);

stat.nErrorId := TO_INT(fbCtrlPid.eErrorId);

// Enable a smooth transition from AUTO to MANUAL mode if needed
IF stat.eCtrlMode = E_METIS_CTRL_MODE.AUTO AND cfg.bSyncManualOut THEN
    ctrl.lrManualOut := stat.lrControllerOut;
END_IF
END_METHOD

METHOD M_ExecuteModes
VAR_INPUT
END_VAR
VAR_INST
    {attribute 'OPC.UA.DA' := '0'}
    fbInputTimer    : TON;
    {attribute 'OPC.UA.DA' := '0'}
    fbSetpointTimer : TON;
    {attribute 'OPC.UA.DA' := '0'}
    fbGetSystemTime : GETSYSTEMTIME;
    {attribute 'OPC.UA.DA' := '0'}
    fileTime        : T_FILETIME;
END_VAR
If stat.eCtrlMode = E_METIS_CTRL_MODE.NONE THEN
    // typical behavior when e.g. a config file did not contain a valid entry
    // To avoid problems, force MANUAL in this case
    stat.eCtrlMode := E_METIS_CTRL_MODE.MANUAL;
END_IF

// check which mode switches are accepted
// (currently very simple, but can be made more complex if needed)
stat.bAcceptCtrlMode_Auto := stat.eCtrlMode = E_METIS_CTRL_MODE.MANUAL
                             AND NOT stat.bError;
stat.bAcceptCtrlMode_Manual := stat.eCtrlMode = E_METIS_CTRL_MODE.AUTO ;

// switch to AUTO / MANUAL mode if acceptable
IF ctrl.eCtrlMode = E_METIS_CTRL_MODE.AUTO AND stat.bAcceptCtrlMode_Auto THEN
    stat.eCtrlMode := E_METIS_CTRL_MODE.AUTO;
ELSIF ctrl.eCtrlMode = E_METIS_CTRL_MODE.MANUAL AND stat.bAcceptCtrlMode_Manual THEN
    stat.eCtrlMode := E_METIS_CTRL_MODE.MANUAL;
END_IF

// switch to engineering ON / OFF mode if acceptable
stat.bEngMode := ctrl.bEngMode;

// switch to manual in any case if the input value is invalid
fbInputTimer(
    IN := (stat.eCtrlMode = E_METIS_CTRL_MODE.AUTO)
          AND (NOT pInputTemp^.stat.bValid),
    PT := DINT_TO_TIME(cfg.nInputTempTimeout));
fbSetpointTimer(
    IN := (stat.eCtrlMode = E_METIS_CTRL_MODE.AUTO)
           AND (NOT pSetpointTemp^.stat.bValid)
           AND cfg.eSetpointSwitch = E_METIS_CTRL_SETPOINT_SWITCH.VARIABLE,
    PT := DINT_TO_TIME(cfg.nSetpointTempTimeout)); 

IF fbInputTimer.Q OR fbSetpointTimer.Q THEN
    // calculate current time here, to avoid dependencies to MAIN.fbServices
    fbGetSystemTime(timeLoDW=>fileTime.dwLowDateTime, timeHiDW=>fileTime.dwHighDateTime );
    stat.sLastForcedManualTime := SYSTEMTIME_TO_STRING(FILETIME_TO_SYSTEMTIME(fileTime));
    IF fbInputTimer.Q THEN
        stat.sLastForcedManualCause := 'Invalid input temperature';
    ELSIF fbSetpointTimer.Q THEN
        stat.sLastForcedManualCause := 'Invalid setpoint temperature';
    ELSE
        stat.sLastForcedManualCause := 'UNKNOWN';
	END_IF
    
    stat.eCtrlMode := E_METIS_CTRL_MODE.MANUAL;
END_IF

// reset any request
ctrl.eCtrlMode := E_METIS_CTRL_MODE.NONE;
END_METHOD

METHOD M_Read_Write_Config
VAR_IN_OUT
    temperatures : FB_METIS_TEMPERATURES;
END_VAR
IF stat.bEngMode THEN
    IF ctrl.bWriteConfig THEN
        
        // update the cfg object
        cfg.sInputTempName      := pInputTemp^.in_sName;
        cfg.sSetpointTempName   := pSetpointTemp^.in_sName;
        cfg.lrFixedSetpoint     := ctrl.lrFixedSetpoint;
        cfg.lrSetpointOffset    := ctrl.lrSetpointOffset; 
        cfg.lrManualOut         := ctrl.lrManualOut;
        
        // write the cfg object
        fbTcConfig.M_WriteConfiguration();
        ctrl.bWriteConfig := FALSE;
                
    ELSIF ctrl.bReadConfig THEN
	
        fbTcConfig.M_ReadConfiguration();
        ctrl.bReadConfig := FALSE;
        
    END_IF
		
END_IF

IF fbTcConfig.bReadingDoneFlag THEN
	M_ConfigReadingFinished(
        bError := fbTcConfig.bReadError,
        temperatures := temperatures);
END_IF
END_METHOD

METHOD M_Set_SetPoint
VAR_INPUT
	m_eSetpointType:		E_METIS_CTRL_SETPOINT_SWITCH:=E_METIS_CTRL_SETPOINT_SWITCH.FIXED;
	m_pSetpointTemp: 		POINTER TO FB_METIS_TEMPERATURE;
	m_lrSetpointOffset: 	LREAL := 0.0;
	m_lrFixedSetpoint:	LREAL;
END_VAR

// Set point type 
cfg.eSetpointSwitch := m_eSetpointType;
// Variable setpoint
stat.lrActVariableSetpoint := m_pSetpointTemp^.stat.lrTempK;
ctrl.lrSetpointOffset:= m_lrSetpointOffset;
// Fixed setpoint
ctrl.lrFixedSetpoint := m_lrFixedSetpoint;
END_METHOD

METHOD M_SetDisable
VAR_INPUT
END_VAR

cfg.bEnabled := FALSE;
ctrl.eCtrlMode := E_METIS_CTRL_MODE.MANUAL;
END_METHOD

METHOD M_SetEnable
VAR_INPUT
END_VAR


cfg.bEnabled := TRUE;
ctrl.eCtrlMode := E_METIS_CTRL_MODE.AUTO;
END_METHOD

METHOD M_Startup : BOOL
VAR_INPUT
END_VAR
VAR_INST
	{attribute 'OPC.UA.DA' := '0'}
    startupTimer : TON;
END_VAR
startupTimer(IN := TRUE, PT := DINT_TO_TIME(cfg.nStartupTimeout));

IF NOT stat.bStarted THEN
    
    IF startupTimer.Q 
       OR (pInputTemp^.stat.bValid
           AND (pSetpointTemp^.stat.bValid 
                OR cfg.eSetpointSwitch = E_METIS_CTRL_SETPOINT_SWITCH.FIXED)) THEN
        stat.bStarted := TRUE; 
    END_IF
END_IF
END_METHOD

METHOD M_UpdateAlarms
VAR_INPUT
END_VAR
VAR
	stEventEntry : TcEventEntry;
	sText : STRING;
END_VAR
//
// Set / clear alarms
//

// Input temperature / process variable is invalid.
fbAlarmHandler.M_UpdateAlarm(
    in_bCondition    := cfg.bEnabled
                        AND stat.bStarted
                        AND (ctrl.nInputTempIndex <> 0)
                        AND (NOT stat.bActInputValid),
    in_nIndex        := 0,
    in_strEventEntry := Tc_Events.METISCryoPIDCtrlEventClass.InputTemperatureInvalid
);


// Variable setpoint temperature is invalid.
fbAlarmHandler.M_UpdateAlarm(
    in_bCondition    := cfg.bEnabled
                        AND stat.bStarted
                        AND (cfg.eSetpointSwitch = E_METIS_CTRL_SETPOINT_SWITCH.VARIABLE)
                        AND (ctrl.nSetpointTempIndex <> 0)
                        AND (NOT stat.bActVariableSetpointValid),
    in_nIndex        := 1,
    in_strEventEntry := Tc_Events.METISCryoPIDCtrlEventClass.VariableSetpointInvalid
);


// Controller was forced to manual mode.
fbAlarmHandler.M_UpdateAlarm(
    in_bCondition    := cfg.bEnabled
                        AND stat.bStarted
                        AND stat.bCtrlModeIsManual
                        AND (stat.sLastForcedManualCause <> ''),
    in_nIndex        := 2,
    in_strEventEntry := Tc_Events.METISCryoPIDCtrlEventClass.ControllerForcedManual
);


// PID function block error.
fbAlarmHandler.M_UpdateAlarm(
    in_bCondition    := cfg.bEnabled
                        AND stat.bStarted
                        AND fbCtrlPid.bError,
    in_nIndex        := 3,
    in_strEventEntry := Tc_Events.METISCryoPIDCtrlEventClass.PidBlockError
);


// Ramp function block error.
fbAlarmHandler.M_UpdateAlarm(
    in_bCondition    := cfg.bEnabled
                        AND stat.bStarted
                        AND ramp.stat.bError,
    in_nIndex        := 4,
    in_strEventEntry := Tc_Events.METISCryoPIDCtrlEventClass.RampBlockError
);


//
// Handle alarms
//
fbAlarmHandler(stAlarms := stat.stAlarms);

fbAlarmHandler.M_ProcessAlarms(
    arrEventEntry := arrEventEntry,
    sEventString  := in_sName
);
END_METHOD

METHOD M_UpdateStatus
VAR_INPUT
END_VAR
ctrl.nInputTempIndex := TO_INT(ctrl.eInputTempIndex);
ctrl.nSetpointTempIndex := TO_INT(ctrl.eVariableSetpointIndex);

// Alarm Handeling
sInstanceName := fbAlarmHandler.sInstanceName;
sEventClassName := fbAlarmHandler.sEventClassName;
IF bConfirmAllAlarms THEN
	bConfirmAllAlarms := FALSE;
	fbAlarmHandler.M_ConfirmAllAlarms();
END_IF

// update some more stat variables
stat.bSetpointSwitchIsFixed := cfg.eSetpointSwitch = E_METIS_CTRL_SETPOINT_SWITCH.FIXED;
stat.bSetpointSwitchIsVariable := cfg.eSetpointSwitch = E_METIS_CTRL_SETPOINT_SWITCH.VARIABLE;
stat.bCtrlModeIsAuto := stat.eCtrlMode = E_METIS_CTRL_MODE.AUTO;
stat.bCtrlModeIsManual := stat.eCtrlMode = E_METIS_CTRL_MODE.MANUAL;
stat.bActInputValid := (ctrl.nInputTempIndex <> 0) AND pInputTemp^.stat.bValid;
stat.bActVariableSetpointValid := (ctrl.nSetpointTempIndex <> 0) AND pSetpointTemp^.stat.bValid;

// update the textual status, and the bError and bWarning flags
IF NOT cfg.bEnabled THEN
    stat.sStatus := 'Disabled';
    stat.bError := FALSE;
ELSIF NOT stat.bStarted THEN
    stat.sStatus := 'Initializing';
ELSIF ctrl.nInputTempIndex = 0 THEN
    stat.sStatus := 'No input temperature configured';
    stat.bError := TRUE;
ELSIF NOT pInputTemp^.stat.bValid THEN
    stat.sStatus := 'Invalid input temperature';
    stat.bError := TRUE;
ELSIF      cfg.eSetpointSwitch = E_METIS_CTRL_SETPOINT_SWITCH.VARIABLE 
       AND ctrl.nSetpointTempIndex = 0 THEN
    stat.sStatus := 'No variable setpoint configured';
    stat.bError := TRUE;
ELSIF      cfg.eSetpointSwitch = E_METIS_CTRL_SETPOINT_SWITCH.VARIABLE 
       AND NOT pSetpointTemp^.stat.bValid THEN
    stat.sStatus := 'Invalid variable setpoint';
    stat.bError := TRUE;
ELSIF fbCtrlPid.bError THEN
    stat.sStatus := CONCAT('PID block error ', INT_TO_STRING(TO_INT(fbCtrlPid.eErrorId)));
    stat.bError := TRUE;
ELSIF ramp.stat.bError THEN
    stat.sStatus := CONCAT('Ramp block error ', INT_TO_STRING(TO_INT(ramp.stat.eErrorId)));
    stat.bError := TRUE;
ELSIF stat.eCtrlMode = E_METIS_CTRL_MODE.MANUAL THEN
    stat.bError := FALSE;
    stat.bWarning := FALSE;
    IF stat.bEngMode THEN
        stat.sStatus := 'MANUAL (ENG MODE)';
    ELSE
        stat.sStatus := 'MANUAL';
	END_IF
ELSIF stat.eCtrlMode = E_METIS_CTRL_MODE.AUTO THEN
    stat.bError := FALSE;
    stat.bWarning := FALSE;
    IF stat.bEngMode THEN
        stat.sStatus := 'AUTO (ENG MODE)';
    ELSE
        stat.sStatus := 'AUTO';
	END_IF
ELSE
    stat.bError := FALSE;
    stat.bWarning := TRUE;
    stat.sStatus := 'UNKNOWN STATUS';
END_IF

stat.bValid := NOT (stat.bError OR stat.bWarning);
END_METHOD

METHOD M_UpdateTempPointers
VAR_INPUT
END_VAR
VAR_IN_OUT
    temperatures : FB_METIS_TEMPERATURES;
END_VAR
VAR 
    i : INT;
END_VAR
pInputTemp    := temperatures.all_temperatures[ctrl.nInputTempIndex];
pSetpointTemp := temperatures.all_temperatures[ctrl.nSetpointTempIndex];
END_METHOD

END_FUNCTION_BLOCK

// POUs/XML_Cfg_Read_Write/FB_READ_WRITE_METIS_CTRL_DT670_CFG
FUNCTION_BLOCK FB_READ_WRITE_METIS_CTRL_DT670_CFG EXTENDS FB_READ_WRITE_CONFIG_BASE
VAR_INPUT
	in_sTempCtrlName:	T_MaxString;
END_VAR
VAR_IN_OUT
	Temp_Ctrl_Config:   T_METIS_CTRL_LOOP_CFG;
END_VAR

SUPER^(
    in_sEntryName  := in_sTempCtrlName,
    in_sSubFolder  := 'Temperature_Control\',
    in_sXPath      := '/Temperature_Control_Configuration/',
    in_pSymAddr    := ADR(Temp_Ctrl_Config),
    in_cbSymSize   := SIZEOF(Temp_Ctrl_Config));

END_FUNCTION_BLOCK

// POUs/XML_Cfg_Read_Write/FB_READ_WRITE_CONFIG_BASE
FUNCTION_BLOCK FB_READ_WRITE_CONFIG_BASE
VAR_INPUT
    in_sEntryName:  T_MaxString := 'Example';   // No slashes!
    in_sSubFolder:  T_MaxString := 'Example\';  // <FolderName>\   (note the last backslash!)
	in_sXPath:      T_MaxString := '/Example/'; // Include a leading and trailing forward slash!
    in_pSymAddr:    PVOID;                      // pointer to the object to store
    in_cbSymSize:   UDINT;                      // SIZEOF the object to store
END_VAR
VAR_OUTPUT
END_VAR
VAR
    // total file path (to be concatenated with the subfolder)
	sFilePath:		T_MaxString := 'C:\Users\Administrator\Desktop\METIS_Cryo_Config_Files\';
    sXPath:         T_MaxString;
    
    // XML function blocks
	fbXmlSrvWrite: 	FB_XmlSrvWrite;
	fbXmlSrvRead:	FB_XmlSrvRead;
	
    // configuration flag
	bConfigured:    BOOL := FALSE;
    
    // state machines
	nWriteState:    INT := 0;
	nReadState:     INT := 0;
    
    // triggers (set by M_ReadConfiguration() and M_WriteConfiguration())
	bExecuteRead:	BOOL := FALSE;
	bExecuteWrite:	BOOL := FALSE;
	
END_VAR
VAR_OUTPUT
	nReadErrorCode:	    UDINT;
	{attribute 'TcHmiSymbol.Show'}
	{attribute 'TcHmiSymbol.ReadOnly'}
	sReadError:         STRING;
    bReadError:         BOOL;
	{attribute 'TcHmiSymbol.Show'}
	{attribute 'TcHmiSymbol.ReadOnly'}
	bReading:           BOOL;
    bReadingDoneFlag:   BOOL;
    
	nWriteErrorCode:    UDINT;
	{attribute 'TcHmiSymbol.Show'}
	{attribute 'TcHmiSymbol.ReadOnly'}
	sWriteError:        STRING;
    bWriteError:        BOOL;
	{attribute 'TcHmiSymbol.Show'}
	{attribute 'TcHmiSymbol.ReadOnly'}
	bWriting:           BOOL;
    bWritingDoneFlag:   BOOL;
END_VAR

M_Configure();

CASE nReadState OF
    0:	
        IF bExecuteRead THEN
            bExecuteRead := FALSE;
            nReadState := 10;
            nReadErrorCode := 0;
            sReadError := 'Reading';
            bReadError := FALSE;
            bReading := TRUE;
            bReadingDoneFlag := FALSE;
		END_IF

    10:
        // execute a rising edge
        fbXmlSrvRead(
            nMode       := XMLSRV_SKIPMISSING,
            pSymAddr	:= in_pSymAddr,
            cbSymSize	:= in_cbSymSize, 
            sFilePath	:= sFilePath,
            sXPath	    := sXPath,
            tTimeout    := T#5s, // tTimeout    := T#30s,
            bExecute	:= FALSE
        );
        fbXmlSrvRead(bExecute := TRUE);
        
        IF fbXmlSrvRead.bError THEN
            nReadState := 900;
        ELSIF fbXmlSrvRead.bBusy THEN
            nReadState := 20;
        END_IF
    20:
        // keep on executing the read FB 
        fbXmlSrvRead(bExecute := TRUE);
        IF fbXmlSrvRead.bError THEN
            nReadState := 900;
        ELSIF NOT fbXmlSrvRead.bBusy THEN
            // done reading!
            nReadState := 1000;
        END_IF
    900:
        nReadErrorCode := fbXmlSrvRead.nErrId;	
        bReading := FALSE;
        bReadingDoneFlag := TRUE;
        bReadError := TRUE;
        sReadError := M_GetErrorString(nReadErrorCode);
        nReadState := 0;
    1000:
        nReadErrorCode := 0;
        sReadError := 'OK';
        bReading := FALSE;
        bReadingDoneFlag := TRUE;
        bReadError := FALSE;
        nReadState := 0;
END_CASE


CASE nWriteState OF
    0:	
        IF bExecuteWrite THEN
            bExecuteWrite := FALSE;
            nWriteState := 10;
            nWriteErrorCode := 0;
            sWriteError := 'Writing';
            bWriteError := FALSE;
            bWriting := TRUE;
            bWritingDoneFlag := FALSE;
		END_IF
		
    10:
        // execute a rising edge
        fbXmlSrvWrite(
            nMode       := XMLSRV_ADDMISSING, 
            pSymAddr    := in_pSymAddr,
            cbSymSize   := in_cbSymSize, 
            sFilePath   := sFilePath, 
            sXPath      := sXPath, 
            bExecute    := FALSE, 
            tTimeout    := T#30S);	// tTimeout    := T#5s 
        fbXmlSrvWrite(bExecute := TRUE);
        
        IF fbXmlSrvWrite.bError THEN
            nWriteState := 900;
        ELSIF fbXmlSrvWrite.bBusy THEN
            nWriteState := 20;
        END_IF
    20:
        // keep on executing the write FB 
        fbXmlSrvWrite(bExecute := TRUE);
        IF fbXmlSrvWrite.bError THEN
            nWriteState := 900;
        ELSIF NOT fbXmlSrvWrite.bBusy THEN
            // done reading!
            nWriteState := 1000;
        END_IF
    900:
        nWriteErrorCode := fbXmlSrvWrite.nErrId;	
        bWriting := FALSE;
        bWritingDoneFlag := TRUE;
        bWriteError := TRUE;
        sWriteError := M_GetErrorString(nWriteErrorCode);
        nWriteState := 0;
    1000:
        nWriteErrorCode := 0;
        sWriteError := 'OK';
        bWriting := FALSE;
        bWritingDoneFlag := TRUE;
        bWriteError := FALSE;
        nWriteState := 0;
END_CASE

PROPERTY bIsReading : BOOL
GET
bIsReading := bReading;
END_GET
END_PROPERTY

PROPERTY bIsWriting : BOOL
GET
bIsWriting := bWriting;
END_GET
END_PROPERTY

METHOD M_ClearReadingDoneFlag
VAR_INPUT
END_VAR
bReadingDoneFlag := FALSE;
END_METHOD

METHOD M_ClearWritingDoneFlag
VAR_INPUT
END_VAR
bWritingDoneFlag := FALSE;
END_METHOD

METHOD M_Configure
VAR_INPUT
END_VAR

IF NOT bConfigured THEN
	
sFilePath := CONCAT(sFilePath, CONCAT(in_sSubFolder, CONCAT(in_sEntryName, '.xml')));
sXPath := CONCAT(in_sXPath, in_sEntryName);

bConfigured := TRUE;

ELSE
	RETURN;
END_IF
END_METHOD

METHOD M_GetErrorString : STRING
VAR_INPUT
    nErrorCode : UDINT;
END_VAR
CASE nErrorCode OF
    6:
        M_GetErrorString := 'XML server not running';
    1804:
        M_GetErrorString := 'File not found';
    ELSE
        M_GetErrorString := CONCAT('Error ', UDINT_TO_STRING(nWriteErrorCode));
END_CASE
END_METHOD

METHOD M_ReadConfiguration
VAR_INPUT
END_VAR
bReadingDoneFlag := FALSE;
bExecuteRead := TRUE;
END_METHOD

METHOD M_WriteConfiguration
VAR_INPUT
END_VAR
bWritingDoneFlag := FALSE;
bExecuteWrite := TRUE;
END_METHOD

END_FUNCTION_BLOCK

// POUs/Control/Control/FB_METIS_CTRL_RAMP_GENERATOR
FUNCTION_BLOCK FB_METIS_CTRL_RAMP_GENERATOR
VAR_INPUT
	{attribute 'OPC.UA.DA' := '0'}
	in_bEnable										: BOOL ;
	{attribute 'OPC.UA.DA' := '0'}
	in_fRampSetPoint								: LREAL;
	{attribute 'OPC.UA.DA' := '0'}
	in_fStartPoint									: LREAL;	// The start point of the ramp (the current actual value)
	{attribute 'OPC.UA.DA' := '0'}
	in_fRampUp_Rate									: LREAL;
	{attribute 'OPC.UA.DA' := '0'}
	in_fRampDown_Rate								: LREAL;
	
END_VAR
VAR_OUTPUT
	{attribute 'OPC.UA.DA' := '0'}
	out_fRampValue									: LREAL;
END_VAR
VAR
	(*Ramp control parameter*)
	ctrl											: T_METIS_CTRL_RAMP_CTRL;

	(* function block *)
	{attribute 'OPC.UA.DA' := '0'}
	fbCTRL_RAMP_GENERATOR							: FB_CTRL_RAMP_GENERATOR;
	{attribute 'OPC.UA.DA' := '0'}
	stCTRL_RAMP_GENERATOR_PARAMS					: ST_CTRL_RAMP_GENERATOR_PARAMS;

	(* Status *)
	stat											: T_METIS_CTRL_RAMP_STAT;
	
    // outputs that can be used for linking
	{attribute 'OPC.UA.DA' := '0'}
    q_lrValue   AT %Q*: LREAL;
	{attribute 'OPC.UA.DA' := '0'}
	q_bToggle   AT %Q*: BOOL;
	{attribute 'OPC.UA.DA' := '0'}
    q_bValid    AT %Q*: BOOL;
    
	{attribute 'OPC.UA.DA' := '0'}
    fbToggleTimer   : TON; 
END_VAR

// Configuration 



M_Configure();


ctrl.RampUp_Rate := in_fRampUp_Rate;
ctrl.RampDown_Rate := in_fRampDown_Rate;

//ctrl.fTarget := in_fRampSetPoint;
stCTRL_RAMP_GENERATOR_PARAMS.fVeloPos			:= ctrl.RampUp_Rate / 60.0; (* 1/60 to convert into units per second *)
stCTRL_RAMP_GENERATOR_PARAMS.fVeloNeg			:= ctrl.RampDown_Rate / 60.0; (* 1/60 to convert into units per second *)


// Execute Controller
M_ExecuteController();

out_fRampValue := stat.fOut;

// update the outputs
fbToggleTimer(IN := (NOT fbToggleTimer.Q) AND in_bEnable, PT := T#1s, Q => q_bToggle);
q_lrValue := stat.fOut;
q_bValid := in_bEnable;

METHOD M_Configure : BOOL
VAR_INPUT
END_VAR



IF in_bEnable THEN
	ctrl.bEnable	:=	TRUE;
ELSE
	ctrl.bEnable	:=	FALSE;
END_IF




IF NOT stat.bConfigured	THEN

(* init parameter struct *)
	stCTRL_RAMP_GENERATOR_PARAMS.tTaskCycleTime		:= T#10MS;
	stCTRL_RAMP_GENERATOR_PARAMS.tCtrlCycleTime		:= T#10MS;
	
	(* reset the init flag *)
	//ctrl.bInit							:= FALSE;
	
	stat.bConfigured	:= TRUE;
ELSE
	RETURN;	// Nothing to do any more
END_IF
END_METHOD

METHOD M_ExecuteController : BOOL
VAR_INPUT
END_VAR
ctrl.fStart := in_fStartPoint;

(* call function block *)
fbCTRL_RAMP_GENERATOR(				bEnable					:= ctrl.bEnable,
									fStart					:= ctrl.fStart,
									fTarget					:= in_fRampSetPoint,//ctrl.fTarget,
									stParams				:= stCTRL_RAMP_GENERATOR_PARAMS,
									fOut					=> stat.fOut,
									bValueReached			=> stat.bValueReached,
									bError					=> stat.bError,
									eErrorId				=> stat.eErrorId);
END_METHOD

END_FUNCTION_BLOCK

// POUs/MAIN
PROGRAM MAIN
VAR
	

	fbServices : FB_SERVICES;
		{attribute 'TcHmiSymbol.Show'}
	met_cryo_ctrl	:	FB_METIS_CRYO_CTRL;
END_VAR



fbServices();

met_cryo_ctrl();

END_PROGRAM

// POUs/Services/FB_SERVICES
FUNCTION_BLOCK FB_SERVICES
VAR_INPUT
END_VAR
VAR_OUTPUT
END_VAR
VAR    
    // Let's always link the EtherCAT DevState, so that 
    // we always have one sync variable (even if all subsystems are disabled)
    {attribute 'TcLinkTo' := 'TIID^Device 1 (EtherCAT)^Inputs^DevState'}
	i_nDevState AT %I* : UINT;
    
    {attribute 'TcLinkTo' := '.i_inTime             := TIID^Device 1 (EtherCAT)^PLC (EK1200)^PTP (EL6688)^  External Sync^Internal time stamp;
                              .i_exTime             := TIID^Device 1 (EtherCAT)^PLC (EK1200)^PTP (EL6688)^  External Sync^External time stamp;
                              .i_dc2TcOffset        := TIID^Device 1 (EtherCAT)^InfoData^DcToTcTimeOffset;
                              .i_dc2ExtOffset       := TIID^Device 1 (EtherCAT)^InfoData^DcToExtTimeOffset;
                              .i_extDevNotConnected := TIID^Device 1 (EtherCAT)^PLC (EK1200)^PTP (EL6688)^  External Sync^External device not connected;
                              .i_AdsAddr            := TIID^Device 1 (EtherCAT)^PLC (EK1200)^PTP (EL6688)^InfoData^AdsAddr;
                              .i_exNtpExtTime       := TIRC^TcCOM Objects^NtpProvider^Outputs^nExtTime;
                              .i_exNtpSysTime       := TIRC^TcCOM Objects^NtpProvider^Outputs^nSysTime;
                              .i_exNtpExtOffset     := TIRC^TcCOM Objects^NtpProvider^Outputs^nSysToExtTimeOffset;
                              .i_NtpConnected       := TIRC^TcCOM Objects^NtpProvider^Diagnostic^bIsConnected;
                              .i_exNtpSynchronized  := TIRC^TcCOM Objects^NtpProvider^Diagnostic^bIsSynchronized'}
    fbTime : FB_TIME;

END_VAR

fbTime();

END_FUNCTION_BLOCK

// POUs/System/FB_METIS_CRYO_CTRL

FUNCTION_BLOCK FB_METIS_CRYO_CTRL
VAR_INPUT
	in_sName:	STRING := 'METIS_CRYO_CTRL';	// Control System name
END_VAR
VAR
	///////////////////////////
	// User Management
	///////////////////////////	
	current_user:		WSTRING;

	///////////////////////////
	// Configuration parameters
	///////////////////////////
		{attribute 'TcHmiSymbol.Show'}
	cfg:	T_METIS_CRYO_CFG;
	
	/////////////////////
	// Control parameters
	/////////////////////
	{attribute 'TcHmiSymbol.Show'}
	ctrl:	T_METIS_CRYO_CTRL;

	/////////////////////
	// Status parameters
	/////////////////////
		{attribute 'TcHmiSymbol.Show'}
	stat:	T_METIS_CRYO_STAT;
	
	/////////////////////
	// System interlocks
	/////////////////////
	{attribute 'TcHmiSymbol.Show'}
	interlocks:	T_METIS_CRYO_INTERLOCKS;

	/////////////////////
	// Debug parameters
	/////////////////////
	debug:	T_METIS_CRYO_DEBUG;

	/////////////////////
	// System Triggers
	/////////////////////
	triggers:	T_METIS_CRYO_TRIGGERS;

	/////////////////////
	// System Events
	/////////////////////
		{attribute 'TcHmiSymbol.Show'}
	events:	T_METIS_CRYO_EVENTS;
	
	/////////////////////
	// Cryo System logs
	/////////////////////
			{attribute 'TcHmiSymbol.Show'}
	logs:	FB_CRYO_FUNCTION_LOG;

	/////////////////////
	// Local variables
	/////////////////////
	
	////////////////////////////////////////////////
	////             Sensors
	////////////////////////////////////////////////
	
	
	/////////////////////////////////////////////////////////
	////                  Temperatures
	/////////////////////////////////////////////////////////
	{attribute 'OPC.UA.DA' := '1'}
		{attribute 'TcHmiSymbol.Show'}
	met_temp:				FB_METIS_TEMPERATURES;  // All temperature sensors
	
	/////////////////////////////////////////////////////////
	////                  Temperature control
	/////////////////////////////////////////////////////////
	{attribute 'OPC.UA.DA' := '1'}
		{attribute 'TcHmiSymbol.Show'}
	met_tctrl:              FB_METIS_TCTRL; // All temperature control loops
    
    /////////////////////////////////////////////////////////
	////                  Heaters
	/////////////////////////////////////////////////////////
	{attribute 'OPC.UA.DA' := '1'}
		{attribute 'TcHmiSymbol.Show'}
	met_heaters:			FB_METIS_HEATERS; // All METIS heaters
	
	
	/////////////////////////////////////////////////////////
	////                  Relative Humidities
	/////////////////////////////////////////////////////////
	{attribute 'OPC.UA.DA' := '1'}
		{attribute 'TcHmiSymbol.Show'}
	met_rh:				FB_METIS_RH;  // All relative humidities
    
    /////////////////////////////////////////////////////////
	////                  Voters
	/////////////////////////////////////////////////////////
	{attribute 'OPC.UA.DA' := '1'}
		{attribute 'TcHmiSymbol.Show'}
    met_voters : FB_METIS_VOTERS; // All METIS voters
    
    /////////////////////////////////////////////////////////
	////                  Lakeshores
	/////////////////////////////////////////////////////////
	{attribute 'OPC.UA.DA' := '1'}
		{attribute 'TcHmiSymbol.Show'}
    met_lakeshores : FB_METIS_LAKESHORES; // All METIS lakeshores
    
    /////////////////////////////////////////////////////////
	////                  CCUs
	/////////////////////////////////////////////////////////
	{attribute 'OPC.UA.DA' := '1'}
		{attribute 'TcHmiSymbol.Show'}
    met_ccus : FB_METIS_CCUS; // All METIS Cabinet Control Units
    
	//////////////////////////////////////////////
	//             Routines
	//////////////////////////////////////////////
		{attribute 'TcHmiSymbol.Show'}
	met_evac:				FB_METIS_CRYO_EVAC;
		{attribute 'TcHmiSymbol.Show'}
	met_venting:			FB_METIS_CRYO_VENTING;
		{attribute 'TcHmiSymbol.Show'}
	met_cool_down:			FB_METIS_CRYO_COOL_DOWN;
		{attribute 'TcHmiSymbol.Show'}
	met_anti_fogging:		FB_METIS_CRYO_ANTI_FOGGING;
		{attribute 'TcHmiSymbol.Show'}
	met_warm_up:			FB_METIS_CRYO_WARM_UP;
		{attribute 'TcHmiSymbol.Show'}
	met_regeneration:		FB_METIS_CRYO_REGENERATION;
		{attribute 'TcHmiSymbol.Show'}
	met_power_outage:		FB_METIS_CRYO_POWER_OUTAGE;
		{attribute 'TcHmiSymbol.Show'}
	met_stop_power_outage:	FB_METIS_CRYO_STOP_POWER_OUTAGE;
	
	
	////////////////////
	// Coolant Valves//
	//////////////////
	
	TPC_A:					FB_CRYO_VALVE_CTRL;
	TPC_B:					FB_CRYO_VALVE_CTRL;
	
		// Pointers to valves
	ptrV:	ARRAY [1..2] OF POINTER TO FB_CRYO_VALVE_CTRL;
	// Pointers to valve commands
	ptrVC:	ARRAY [1..2] OF POINTER TO FB_CRYO_CMD_OVERRIDE;
	// Pointers to Enable flags for valves
	ptrEV:	ARRAY [1..2] OF POINTER TO BOOL;	
	
	cmdTPC_A:	FB_CRYO_ACTUATOR_CMD;	// Handling of Valve1 command
	cmdTPC_B:	FB_CRYO_ACTUATOR_CMD;	// Handling of Valve1 command
	
	guiCoolantValveIndex:	UINT := 1;	// Index for Valve Engineering GUI
	
	///////////////////////
	// Ambient Pressure //
	/////////////////////
	
	sensor_AMB_PRESS:			FB_METIS_AMBIENT_PRESSURE_SENSOR;
	
	// Sim ambient Pressure values
	q_nSimAmbPress			AT %Q*:	INT := 14330;
	
	//////////////////////
	// System triggers //
	////////////////////	
	{attribute 'OPC.UA.DA' := '0'}
	trgSystemEnable:		R_TRIG;
	{attribute 'OPC.UA.DA' := '0'}
	trgSystemDisable:		F_TRIG;
	
	{attribute 'OPC.UA.DA' := '0'}
	trgEvacOn:			R_TRIG;
	{attribute 'OPC.UA.DA' := '0'}
	trgEvacOff:			F_TRIG;
	{attribute 'OPC.UA.DA' := '0'}
	trgCool:			R_TRIG;
	{attribute 'OPC.UA.DA' := '0'}
	trgCoolOff:			F_TRIG;
	{attribute 'OPC.UA.DA' := '0'}
	trgWarmup:			R_TRIG;
	{attribute 'OPC.UA.DA' := '0'}
	trgWarmupOff:		F_TRIG;
	{attribute 'OPC.UA.DA' := '0'}
	trgRegeneration:	R_TRIG;
	{attribute 'OPC.UA.DA' := '0'}
	trgRegenerationOff:	F_TRIG;
	{attribute 'OPC.UA.DA' := '0'}
	trgVenting:			R_TRIG;
	{attribute 'OPC.UA.DA' := '0'}
	trgVentingOff:		F_TRIG;
	{attribute 'OPC.UA.DA' := '0'}
	trgPoweroutage:		R_TRIG;
	{attribute 'OPC.UA.DA' := '0'}
	trgPoweroutageOff:	F_TRIG;
	
	{attribute 'OPC.UA.DA' := '0'}
	trgInGoodVaccum:	R_TRIG;
	{attribute 'OPC.UA.DA' := '0'}
	trgInVaccum:	R_TRIG;
	{attribute 'OPC.UA.DA' := '0'}
	trgPressurized:	R_TRIG;
	
	{attribute 'OPC.UA.DA' := '0'}
	trgWarm:	R_TRIG;
	{attribute 'OPC.UA.DA' := '0'}
	trgCold:	R_TRIG;
	
	/////////////////////
	// Local variables
	/////////////////////



	{attribute 'OPC.UA.DA' := '0'}
	timer:		TON;		// Timer for commands
	
	{attribute 'OPC.UA.DA' := '0'}
	ptrLog:		ARRAY [0..9] OF POINTER TO STRING(80);
	{attribute 'OPC.UA.DA' := '0'}
	nLogPos:	INT := -1;
	
	///////////////
	// Simulation///
	//////////////
	
	// Sim venting valves simulation
	
	sim_venting_valves:		FB_SIM_VENTING_VALVES;
	
	// Pre_cooling valve simulation
	
	sim_cool_down_valves:	FB_SIM_PRE_COOLING_VALVES;
	
	// Sim LN2 Sensors
	sim_SHA_LS:	FB_SIM_LN2_SENSOR;
	sim_SHB_LS:	FB_SIM_LN2_SENSOR;
	sim_SHC_LS:	FB_SIM_LN2_SENSOR;
	
	// Sim LN2 Level-control valves
	
	sim_LN2_Valves:	FB_SIM_LN2_LEVEL_VALVES;
	
	
	
	(*Pressure on  sleeves of Pulse Tube Coolers*)
	
	// Pressure transducers
	{attribute 'OPC.UA.DA' := '1'}
	sensor_VAG_PTA:	FB_CRYO_SENSOR_PRESSURE;	// Cooling circuit pressure gauge #1
	{attribute 'OPC.UA.DA' := '1'}
	sensor_VAG_PTB:	FB_CRYO_SENSOR_PRESSURE;	// Cooling circuit pressure gauge #2
	{attribute 'OPC.UA.DA' := '1'}
	sensor_VAG_PTC:	FB_CRYO_SENSOR_PRESSURE;	// Cooling circuit pressure gauge #3
	
	{attribute 'OPC.UA.DA' := '1'}
	VAG_PTA:	FB_CRYO_PRESSURE_VOTE;				// Cooling circuit pressure gauge #1
	{attribute 'OPC.UA.DA' := '1'}
	VAG_PTB:	FB_CRYO_PRESSURE_VOTE;				// Cooling circuit pressure gauge #2
	{attribute 'OPC.UA.DA' := '1'}
	VAG_PTC:	FB_CRYO_PRESSURE_VOTE;				// Cooling circuit pressure gauge #3
	
	// Pressure sensors IDN resistors
	
	nIdnRes_VAG_PTA		AT %I* :INT;
	nIdnRes_VAG_PTB		AT %I* :INT;
	nIdnRes_VAG_PTC		AT %I* :INT;
	
	// Pressure sensor power 24V Dig Out
	
	bPwr_VAG_PTA		AT %Q* :BOOL;
	bPwr_VAG_PTB        AT %Q* :BOOL;
	bPwr_VAG_PTC        AT %Q* :BOOL;
	
	
	// Configure
	
	bConfigured:		BOOL := FALSE;
	
	// Relay ctrl for 230 VAC Power for Valves
	// vaccum branch A valves
	bPwr_PVVAs				AT %Q*	:BOOL := TRUE;  
	bFeedBackPwr_PVVAs		AT %Q*	:BOOL := TRUE;
	// vaccum branch B valves
	bPwr_PVVBs				AT %Q*	:BOOL := TRUE;  
	bFeedBackPwr_PVVBs		AT %Q*	:BOOL := TRUE;
	// Repressurization valves
	bPwr_N2Vs				AT %Q*	:BOOL := TRUE;  
	bFeedBackPwr_N2Vs		AT %Q*	:BOOL := TRUE;
	// Cooling circuit
	bPwr_PVVPs				AT %Q*	:BOOL := TRUE;  
	bFeedBackPwr_PVVPs		AT %Q*	:BOOL := TRUE;
	// 
	
	//////////////////
	///Simulations/// 
	////////////////
	
	sim_regeneration: FB_SIM_REGENERATION;
	
	sim_lrHighestTemp: 			LREAL := 200;
	sim_lrLowestTemp:			LREAL := 200;
	sim_lrCryostatTemp:			LREAL := 200;
	sim_lrRadiationShielsTemp:	LREAL := 200;
	
	sim_lrDewPointTempC:		LREAL := 30;
	sim_lrAmbiantTempC:			LREAL := 30;
	sim_lrWindowMountTempC:		LREAL := 30;
	
	/////////////////////////////
	//// Time (NTP from ICS) /// 
	//////////////////////////

	met_cry_time : FB_TIME;
	
	////////////////////
	//// HMI Screen /// 
	//////////////////

	fuseHMI:			FB_FUSE;
	bHMISwitch AT %I* : BOOL;

	/////////////////////////////
	////     TE2000 HMI		 /// 
	//////////////////////////
// Cryo Pressures
	hmi_pressure_vote_vagf : FB_HMI_CRYO_PRESSURE_VOTE;
	hmi_pressure_vote_vagg : FB_HMI_CRYO_PRESSURE_VOTE;
	
	hmi_pressure_vote_vagg1 : FB_HMI_CRYO_PRESSURE_VOTE;
	hmi_pressure_vote_vagg2 : FB_HMI_CRYO_PRESSURE_VOTE;
	
	hmi_pressure_vote_vagf1 : FB_HMI_CRYO_PRESSURE_VOTE;
	hmi_pressure_vote_vagf2 : FB_HMI_CRYO_PRESSURE_VOTE;
// Pumps
	hmi_pump_tmp_a: FB_HMI_CRYO_PUMP;
	hmi_pump_pvp_a: FB_HMI_CRYO_PUMP;
	
	hmi_pump_tmp_b: FB_HMI_CRYO_PUMP;
	hmi_pump_pvp_b: FB_HMI_CRYO_PUMP;
	
// Branch A
	hmi_valve_pvv1_a: FB_HMI_CRYO_VALVE;
	hmi_valve_pvv2_a: FB_HMI_CRYO_VALVE;
	hmi_valve_pvv3_a: FB_HMI_CRYO_VALVE;
	hmi_valve_pvv4_a: FB_HMI_CRYO_VALVE;
	hmi_valve_GBV_a:  FB_HMI_CRYO_VALVE;
	
	hmi_pressure_vote_vag1_a : FB_HMI_CRYO_PRESSURE_VOTE;
	hmi_pressure_vote_vag2_a : FB_HMI_CRYO_PRESSURE_VOTE;
	hmi_pressure_vote_vag3_a : FB_HMI_CRYO_PRESSURE_VOTE;
	
// Branch B
	hmi_valve_pvv1_b: FB_HMI_CRYO_VALVE;
	hmi_valve_pvv2_b: FB_HMI_CRYO_VALVE;
	hmi_valve_pvv3_b: FB_HMI_CRYO_VALVE;
	hmi_valve_pvv4_b: FB_HMI_CRYO_VALVE;
	hmi_valve_GBV_b:  FB_HMI_CRYO_VALVE;
	
	hmi_pressure_vote_vag1_b : FB_HMI_CRYO_PRESSURE_VOTE;
	hmi_pressure_vote_vag2_b : FB_HMI_CRYO_PRESSURE_VOTE;
	hmi_pressure_vote_vag3_b : FB_HMI_CRYO_PRESSURE_VOTE;

// PreCooling
	hmi_valve_pvv_P1: FB_HMI_CRYO_VALVE;
	hmi_valve_pvv_P2: FB_HMI_CRYO_VALVE;
	hmi_valve_pvv_P3: FB_HMI_CRYO_VALVE;
	
	hmi_pressure_vote_vag_pca : FB_HMI_CRYO_PRESSURE_VOTE;
	hmi_pressure_vote_vag_pcb : FB_HMI_CRYO_PRESSURE_VOTE;
	hmi_pressure_vote_vag_p1 : FB_HMI_CRYO_PRESSURE_VOTE;
	
// Venting valves
	hmi_valve_n2v1: FB_HMI_CRYO_VALVE;
	hmi_valve_n2v2: FB_HMI_CRYO_VALVE;

// Water Cooling Valves
	hmi_valve_tpc_A: FB_HMI_CRYO_VALVE;
	hmi_valve_tpc_B: FB_HMI_CRYO_VALVE;

// LN2 Level Control Valves
	hmi_valve_ln2_StifRingSeg: 		FB_HMI_CRYO_VALVE;
	hmi_valve_ln2_IntermediateSeg: 	FB_HMI_CRYO_VALVE;
	hmi_valve_ln2_BottomSeg: 		FB_HMI_CRYO_VALVE;
	
// HPGs
	hmi_pressure_vote_hpg : FB_HMI_CRYO_PRESSURE_VOTE;
	hmi_pressure_vote_hpg1 : FB_HMI_CRYO_PRESSURE_VOTE;
	hmi_pressure_vote_hpg2 : FB_HMI_CRYO_PRESSURE_VOTE;	
	
// Coolers

	// Sleeves Pressures
	hmi_pressure_vote_vag_pta : FB_HMI_CRYO_PRESSURE_VOTE;
	hmi_pressure_vote_vag_ptb : FB_HMI_CRYO_PRESSURE_VOTE;
	hmi_pressure_vote_vag_ptc : FB_HMI_CRYO_PRESSURE_VOTE;

// LN2 Level Control Valves
	hmi_valve_shav: FB_HMI_CRYO_VALVE;
	hmi_valve_shbv: FB_HMI_CRYO_VALVE;
	hmi_valve_shcv: FB_HMI_CRYO_VALVE;
	

	
END_VAR

VAR CONSTANT
	
	/////////////////////////////
	////     DETECTORS		 /// 
	//////////////////////////

    // --- [6000] Detector Preconditions / Status ---
    E6000_DetectorPoweredOnTooEarly               : UDINT := 6000001; // Detector powered on before reaching allowed working temperature
    E6001_DetectorWorkingTempNotReached           : UDINT := 6000002; // Detector has not yet reached working temperature
    E6002_DetectorFunctionTestActive              : UDINT := 6000003; // Detector quick functionality test active
    E6003_DetectorTemperatureSensorFault          : UDINT := 6000004; // Detector temperature sensor invalid or faulty
    E6004_DetectorReferenceTempSensorFault        : UDINT := 6000005; // Reference temperature sensor for coldest-part comparison invalid
    E6005_DetectorProtectionNotInitialized        : UDINT := 6000006; // Detector protection logic not initialized

    // --- [6100] Detector Temperature Safety Alarms ---
    E6100_DetectorTooColdComparedToCryostat       : UDINT := 6100001; // Detector became the coldest part inside the cryostat
    E6101_DetectorTemperatureTooHigh              : UDINT := 6100002; // Detector temperature > 310 K
    E6102_DetectorCooldownRateTooFast             : UDINT := 6100003; // Detector cooling rate exceeds 1 K/min
    E6103_DetectorWarmupRateTooFast               : UDINT := 6100004; // Detector warm-up rate exceeds 1 K/min
    E6104_DetectorTemperatureChangeTooFast        : UDINT := 6100005; // General detector temperature change exceeds 1 K/min
    E6105_DetectorTemperatureControlFailure       : UDINT := 6100006; // Detector temperature control failed or became unstable
    E6106_DetectorTemperatureRunaway              : UDINT := 6100007; // Detector temperature moved uncontrollably after failure or power event

    // --- [6200] Cool Down Related Detector Errors ---
    E6200_DetectorCooldownStartedTooEarly         : UDINT := 6200001; // Detector cooldown started before cryostat conditions were safe
    E6201_DetectorReachedUnsafeLowTemp            : UDINT := 6200002; // Detector temperature dropped below allowed relationship to surrounding cryostat temperatures
    E6202_DetectorNotProtectedDuringCooldown      : UDINT := 6200003; // Detector protection logic not active during cooldown
    E6203_DetectorEnabledDuringCooldown           : UDINT := 6200004; // Detector electronics enabled during cooldown before allowed temperature

    // --- [6300] Warm Up Related Detector Errors ---
    E6300_DetectorWarmupRampControlFault          : UDINT := 6300001; // Detector warm-up ramp control failed
    E6301_DetectorExceeded80KTransitionRule       : UDINT := 6300002; // Detector transition condition around 80 K not respected
    E6302_DetectorExceeded290KSetpoint            : UDINT := 6300003; // Detector exceeded warm-up target setpoint
    E6303_DetectorNotProtectedDuringWarmup        : UDINT := 6300004; // Detector protection logic not active during warm up

    // --- [6400] Power Failure / Uncontrolled Condition Errors ---
    E6400_PowerFailure_DetectorRampTooFast        : UDINT := 6400001; // Detector temperature changed faster than 1 K/min during power failure
    E6401_CoolingLoss_DetectorRampTooFast         : UDINT := 6400002; // Detector temperature changed faster than 1 K/min after sudden cooling loss
    E6402_TCtrlFailure_DetectorRampTooFast        : UDINT := 6400003; // Detector temperature changed faster than 1 K/min after temperature control failure
    E6403_DetectorProtectionLostDuringPowerEvent  : UDINT := 6400004; // Detector protection unavailable during power failure or recovery

    // --- [6500] Operational / Manual Action Errors ---
    E6500_OperatorEnabledDetectorOutsideLimits    : UDINT := 6500001; // Operator enabled detector outside allowed temperature conditions
    E6501_DetectorQuickTestOutsideSafeLimits      : UDINT := 6500002; // Quick functionality test requested outside safe limits
    E6502_DetectorOperationNotAllowedInState      : UDINT := 6500003; // Detector operation requested in an invalid cryostat state

    // --- [6600] Interlock Violations ---
    E6600_DetectorMustRemainOff                   : UDINT := 6600001; // Detector shall remain switched off under current conditions
    E6601_DetectorEnableBlockedByTemperature      : UDINT := 6600002; // Detector enable blocked because temperature conditions are not safe
    E6602_DetectorEnableBlockedByRampRate         : UDINT := 6600003; // Detector enable blocked because temperature ramp is too fast
    E6603_DetectorEnableBlockedByProtectionFault  : UDINT := 6600004; // Detector enable blocked because detector protection is faulty

    // --- [6700] Protective Action / Recovery Failures ---
    E6700_DetectorFailedToSwitchOff               : UDINT := 6700001; // Detector could not be switched off when protection demanded it
    E6701_DetectorProtectionRecoveryFailed        : UDINT := 6700002; // Detector protection did not recover after fault
    E6702_DetectorAlarmNotCleared                 : UDINT := 6700003; // Detector alarm condition persisted after recovery attempt


    // --- [9900] Warm Pressurized Status Alarms ---
    E9900001_WP_ColdStructureTempTooHigh         : UDINT := 9900001; // Cold structure temperature > 310 K
    E9900002_WP_DetectorTempTooHigh              : UDINT := 9900002; // Detector temperature > 310 K
    E9900003_WP_RadiationShieldTempTooHigh       : UDINT := 9900003; // Radiation shield temperature > 310 K

    // --- [9910] Warm Pressurized Interlocks ---
    E9910001_WP_PrecoolingFillingBlocked         : UDINT := 9910001; // Precooling system filling valves blocked
    E9910002_WP_LN2FillingBlocked                : UDINT := 9910002; // LN2 filling blocked
    E9910003_WP_ICARMotorsBlocked                : UDINT := 9910003; // ICAR motors blocked

    // --- [9901] Warm Vacuum Status Alarms ---
    E9901001_WV_ColdStructureTempTooHigh         : UDINT := 9901001; // Cold structure temperature > 310 K
    E9901002_WV_DetectorTempTooHigh              : UDINT := 9901002; // Detector temperature > 310 K
    E9901003_WV_RadiationShieldTempTooHigh       : UDINT := 9901003; // Radiation shield temperature > 310 K
    E9901004_WV_CryostatPressureTooHigh          : UDINT := 9901004; // Cryostat pressure > 1e-4 mbar

    // --- [9902] Cold Status Alarms ---
    E9902001_COLD_CryostatPressureTooHigh        : UDINT := 9902001; // Cryostat pressure > 1e-5 mbar
    E9902002_COLD_ColdStructureTempTooHigh       : UDINT := 9902002; // Cold structure temperature > 75 K
    E9902003_COLD_TemperatureTooLow              : UDINT := 9902003; // Temperature below setpoint - 5 K
    E9902004_COLD_RadiationShieldTempTooHigh     : UDINT := 9902004; // Radiation shield temperature > 100 K
    E9902005_COLD_LN2LevelLowAlarm               : UDINT := 9902005; // LN2 level sensor low alarm triggered
    E9902006_COLD_LN2LevelHighAlarm              : UDINT := 9902006; // LN2 level sensor high alarm triggered
    E9902007_COLD_PrecoolingPressureTooHigh      : UDINT := 9902007; // Pressure in precooling system > 1 mbar

    // --- [9912] Cold Status Interlocks ---
    E9912001_COLD_VentingBlocked                 : UDINT := 9912001; // Venting blocked in cold state
    E9912002_COLD_SorptionHeaterBlocked          : UDINT := 9912002; // Sorption pump heater blocked
    E9912003_COLD_PrecoolingValvesBlocked        : UDINT := 9912003; // Filling and exhaust valves of precooling system blocked

    // --- [9920] Status Detection Errors ---
    E9920001_StatusUndefined                     : UDINT := 9920001; // Instrument status cannot be determined
    E9920002_StatusConflict                      : UDINT := 9920002; // Conflicting status conditions detected
    E9920003_StatusTransitionInvalid             : UDINT := 9920003; // Invalid transition between instrument statuses

END_VAR



M_HMI_Screen_Control();

current_user := VisuElems.CurrentUserName;

M_Configure();


// Simulation
 
{IF defined (V2_SIM)}
	stat.bSimulation := TRUE;
{END_IF}

{IF defined (V1_HW)}
	stat.bSimulation := FALSE;
{END_IF}

	
// venting valves simulation
sim_venting_valves();	

// Pre_cooling valve simulation
sim_cool_down_valves();

// Sim LN2 Level Sensors and Valves
sim_SHA_LS();
sim_SHB_LS();
sim_SHC_LS();

sim_LN2_Valves();


M_ReadSensors();


// Increment cycle counter
stat.nCycleCounter := stat.nCycleCounter + 1;

////
//// Check for sensor HW errors
////
//M_CheckForSensorErrors();



/////////////////////
//// System Operation
/////////////////////

////
//// Execute Controllers
////
M_ExecuteControllers();


////
//// Capture system commands
////
M_CheckForCommands();


////
//// Perform a safety check
////
//M_SafetyCheck();


M_UpdateStatus();


M_ProcessHmi();

////
//// Execute system state machine
////
M_StateMachine();

METHOD M_Activity_Cold_State : BOOL
VAR_INPUT
END_VAR
ctrl.bSafe_Evac            := TRUE; (*TODO: Check with Werner*)
ctrl.bSafe_Cool_Down       := FALSE; 
ctrl.bSafe_Warm_Up         := TRUE;
ctrl.bSafe_Regeneration    := FALSE;
ctrl.bSafe_Venting         := FALSE;
ctrl.bEnable_Venting       := FALSE;
ctrl.bSafe_Anti_Fogging    := TRUE;

stat.bPermitEvacuationStop := TRUE;


// Handle commands (only WARM_UP allowed in COLD state)
IF ctrl.bExecute THEN
    ctrl.bExecute       := FALSE;
    stat.nLastCommand   := ctrl.nCommand;
    ctrl.nCommand       := E_METIS_CRYO_CTRL_CMD.NONE;

    IF stat.nLastCommand = E_METIS_CRYO_CTRL_CMD.WARM_UP THEN
        logs.M_LogInfo('Warm-Up initiated by operator');
        ctrl.bSafe_Warm_Up := TRUE;

        stat.nState := E_METIS_CRYO_CTRL_STATE.WARMING_UP;
    ELSE
        logs.M_LogWarning('Invalid command received in COLD state: ignored.');
    END_IF

ELSE
    
    met_cool_down.M_Activity_Cold_State();
END_IF

M_SetStatus(stat.nState);
RETURN;



//ctrl.bSafe_Evac 			:= TRUE;
//ctrl.bSafe_Cool_Down 		:= FALSE;
//ctrl.bSafe_Warm_Up 			:= FALSE;
//ctrl.bSafe_Regeneration 	:= FALSE;
//ctrl.bSafe_Venting 			:= FALSE;
//ctrl.bEnable_Venting		:= FALSE;
//ctrl.bSafe_Anti_Fogging		:= TRUE;
//stat.bPermitEvacuationStop 	:= TRUE;

////
//// Only WARM_UP command is allowed in state COLD.

//IF	ctrl.bExecute	THEN
//	ctrl.bExecute		:= FALSE;
//	stat.nLastCommand	:= ctrl.nCommand;
//	ctrl.nCommand		:= E_METIS_CRYO_CTRL_CMD.NONE;
//	IF stat.nLastCommand = E_METIS_CRYO_CTRL_CMD.WARM_UP	THEN
		
//		ctrl.bSafe_Warm_Up := TRUE;
//		IF NOT ctrl.bEnable_Evac THEN 
//			ctrl.bEnable_Evac  := TRUE;
//		END_IF
		
//		logs.M_LogInfo('Warm-Up initiated by operator');
//		stat.nState	:= E_METIS_CRYO_CTRL_STATE.WARMING_UP;
//	END_IF
//ELSE
//	met_cool_down.M_Activity_Cold_State();
//	stat.nState	:= E_METIS_CRYO_CTRL_STATE.COLD;
//END_IF
//M_SetStatus(stat.nState);	
//RETURN;
END_METHOD

METHOD M_Activity_Cooling_Down_State : BOOL
VAR_INPUT
END_VAR

ctrl.bSafe_Evac             := TRUE;
ctrl.bSafe_Cool_Down        := TRUE;
ctrl.bSafe_Warm_Up          := FALSE;
ctrl.bSafe_Regeneration     := FALSE;
ctrl.bSafe_Anti_Fogging     := TRUE;
ctrl.bSafe_Venting          := FALSE;
ctrl.bEnable_Venting        := FALSE;

stat.bPermitEvacuationStop  := FALSE;
 

// Check for Cool-Down is finished (automatically or interupted)
IF trgCoolOFF.Q THEN
	ctrl.bEnable_Cool_Down := FALSE;

	// Status change is already logged by the Cool-Down routine
	IF stat.bOP THEN
		stat.nState := E_METIS_CRYO_CTRL_STATE.COLD;
		logs.M_LogInfo('System is already operational. Transitioning to COLD state.');

	ELSIF stat.bPartiallyCold THEN
		stat.nState := E_METIS_CRYO_CTRL_STATE.PARTIALLY_COLD;
		logs.M_LogInfo('Partial cooldown detected. Transitioning to PARTIALLY_COLD state.');
	ELSIF stat.bWarm THEN
		stat.nState := E_METIS_CRYO_CTRL_STATE.WARM_VACUUM;
		logs.M_LogInfo('Cryostat is warm. Transitioning to WARM_VACUUM.');
	ELSE
		// Undefined thermal status — safety fallback
		logs.M_LogWarning('Cool-Down interrupted but system is in unknown thermal state.');
		stat.nState := E_METIS_CRYO_CTRL_STATE.ERROR;
	END_IF

	M_SetStatus(stat.nState);
	RETURN;
END_IF

// Continue in COOLING_DOWN state
M_SetStatus(stat.nState);
RETURN;
END_METHOD

METHOD M_Activity_Error_State : BOOL
VAR_INPUT
END_VAR
VAR_INST
    ErrorDurationTimer : TON;
    tErrorTimeout      : TIME := T#10M;
    bFirstEntry        : BOOL := TRUE;
END_VAR
IF bFirstEntry THEN
    bFirstEntry := FALSE;
    logs.M_LogWarning('CRYO CONTROL entered ERROR state.');
    //logs.M_LogWarning(CONCAT('Last Error Code: ', INT_TO_STRING(stat.nLastError)));
    logs.M_LogWarning('Operator intervention required. Awaiting reset or auto-clear.');
    ErrorDurationTimer(IN := TRUE, PT := tErrorTimeout);
    stat.sState := 'ERROR: Awaiting Reset or Resolution';
    M_SetStatus(E_METIS_CRYO_CTRL_STATE.ERROR);
    RETURN;
END_IF

// Allow auto-recovery if the error flag cleared elsewhere
IF NOT stat.bError THEN
    logs.M_LogInfo('Auto-cleared: Exiting ERROR state.');
    ErrorDurationTimer(IN := FALSE);
    stat.nState := E_METIS_CRYO_CTRL_STATE.NONE;
    stat.bInitialized := FALSE;
    bFirstEntry := TRUE;
    RETURN;
END_IF

// Operator-triggered reset
IF ctrl.bReset THEN
    logs.M_LogInfo('Operator RESET issued. Recovering system...');
    ctrl.bReset := FALSE;
    ErrorDurationTimer(IN := FALSE);
    stat.nState := E_METIS_CRYO_CTRL_STATE.NONE;
    stat.bInitialized := FALSE;
    bFirstEntry := TRUE;
    RETURN;
END_IF

// Time exceeded in ERROR without resolution
IF ErrorDurationTimer.Q THEN
    logs.M_LogWarning('Prolonged ERROR state. System unresponsive for 10 minutes.');
    // Here you could: Raise a higher-level alarm, write a persistent fault, or notify external system.
    ErrorDurationTimer(IN := FALSE); // Stop timer if one-time use
END_IF

// Stay in ERROR until reset or auto-clear
RETURN;


//	// RESET the controller in order to try to clear error
//	IF ctrl.bReset THEN
//		ctrl.bReset	:= FALSE;	// Clear RESET flag
//		// Goto NONE state
//		stat.nState	:= E_METIS_CRYO_CTRL_STATE.NONE;
//		stat.bInitialized := FALSE;
//		M_SetStatus(stat.nState);	
//	ELSIF NOT stat.bError  THEN
//		// Goto NONE state
//		stat.nState	:= E_METIS_CRYO_CTRL_STATE.NONE;
//		stat.bInitialized := FALSE;
//		M_SetStatus(stat.nState);	
//	END_IF
//	RETURN;
END_METHOD

METHOD M_Activity_None : BOOL
VAR_INPUT
END_VAR
VAR_INST
    bStarted:           BOOL := FALSE;
    Start_Timer:        TON;


    Init_Timer:         TON;

    bLogToggle:         BOOL := FALSE;

    nNoneSubState:      INT := 0; 

	
	{IF defined (V1_HW)}
		tStart_TimeOut:     TIME := T#90S;
    	tInit_TimeOut:      TIME := cfg.tInitTimeOut;
	{END_IF}
 
	{IF defined (V2_SIM)}
		tStart_TimeOut:     TIME := T#10S;
    	tInit_TimeOut:      TIME := T#20S;
	{END_IF}
	
END_VAR
CASE nNoneSubState OF


        0: // On power-up: start initial wait

            IF NOT bStarted THEN
                bStarted := TRUE;
                logs.M_LogInfo('Cryo controller powered up. Waiting for system stabilization...');
				stat.sState := 'Powered ON: Stabilizing...';
                RETURN;
            END_IF
			
			Start_Timer(IN := TRUE, PT := tStart_TimeOut);
		
			IF Start_Timer.Q THEN
				Start_Timer(IN := FALSE); // stop the timer
				nNoneSubState := 10;
			END_IF
		
			RETURN;


        10: // After wait, check if system is not warm pressurized

            M_GetState(); // Detect the actual system condition

            IF stat.nState <> E_METIS_CRYO_CTRL_STATE.WARM_PRESS THEN
                logs.M_LogWarning('System is not in warm pressurized state. Stabilizing conditions...');
                M_Activity_Stabilize_Cryostat_Conditions();
            END_IF

            nNoneSubState := 20;
			stat.nState := E_METIS_CRYO_CTRL_STATE.NONE;
			stat.bInitialized := FALSE;
            RETURN;


        20: // Wait for operator to enable the controller

//            IF ctrl.bEnable THEN

                IF NOT bLogToggle THEN
                    logs.M_LogInfo('System enabled by operator.');
                    logs.M_LogInfo('Initializing cryo control...');
                    bLogToggle := TRUE;
                END_IF

                Init_Timer(IN := TRUE, PT := tInit_TimeOut);

                IF Init_Timer.Q THEN
                    Init_Timer(IN := FALSE);
                    M_GetState(); // Transition to next valid control state
                    RETURN;
                ELSE
                    stat.sState := 'Initializing Controller...';
                    stat.bActive := TRUE;

                    IF trgSystemDisable.Q THEN
                        logs.M_LogWarning('Cryo control initialization aborted by operator.');
                        stat.sState := 'Initialization Aborted';
                        stat.bActive := FALSE;
                        ctrl.nCommand := E_METIS_CRYO_CTRL_CMD.NONE;
                        Init_Timer(IN := FALSE);
                        RETURN;
                    END_IF

                    RETURN;
                END_IF

//            ELSE
//                stat.sState := 'Inactive: Enable When Ready';
//                stat.bActive := FALSE;
//                RETURN;
//            END_IF

    END_CASE
END_METHOD

METHOD M_Activity_Partial_Vacuum_State : BOOL
VAR_INPUT
END_VAR
ctrl.bSafe_Evac 		:= TRUE;
ctrl.bSafe_Cool_Down 	:= FALSE;
ctrl.bSafe_Warm_Up		:= FALSE;
ctrl.bSafe_Regeneration := TRUE;
ctrl.bSafe_Venting 		:= TRUE;


IF ctrl.bExecute THEN
	ctrl.bExecute      := FALSE;
	stat.nLastCommand  := ctrl.nCommand;
	ctrl.nCommand      := E_METIS_CRYO_CTRL_CMD.NONE;

	CASE stat.nLastCommand OF
		E_METIS_CRYO_CTRL_CMD.VENT:
			logs.M_LogInfo('VENTING initiated by operator.');
			stat.nState := E_METIS_CRYO_CTRL_STATE.VENTING;

		E_METIS_CRYO_CTRL_CMD.NONE:
			// no-op, already handled by reset
			;

		ELSE
			logs.M_LogWarning(CONCAT('Command not allowed in Partial Vacuum state: ', TO_STRING(stat.nLastCommand)));

	END_CASE

	RETURN;
END_IF

// Check if target vacuum level has been reached
IF stat.bInVacuum OR stat.bInGoodVacuum THEN
	logs.M_LogInfo('Target vacuum level achieved. Transitioning to WARM_VACUUM.');
	stat.nState := E_METIS_CRYO_CTRL_STATE.WARM_VACUUM;
	RETURN;
END_IF


M_SetStatus(stat.nState);
RETURN;
END_METHOD

METHOD M_Activity_Partially_Cold_State : BOOL
VAR_INPUT
END_VAR

ctrl.bSafe_Evac            := TRUE;
ctrl.bSafe_Cool_Down       := TRUE;
ctrl.bSafe_Warm_Up         := TRUE;
ctrl.bSafe_Regeneration    := FALSE;
ctrl.bSafe_Anti_Fogging    := TRUE;
ctrl.bSafe_Venting         := FALSE;
ctrl.bEnable_Venting       := FALSE;

stat.bPermitEvacuationStop := FALSE;


IF ctrl.bExecute THEN
    ctrl.bExecute       := FALSE;
    stat.nLastCommand   := ctrl.nCommand;
    ctrl.nCommand       := E_METIS_CRYO_CTRL_CMD.NONE;

    CASE stat.nLastCommand OF

        E_METIS_CRYO_CTRL_CMD.COOL:
            logs.M_LogInfo('Cool-Down re-initiated by operator from PARTIALLY_COLD state');
            stat.nState := E_METIS_CRYO_CTRL_STATE.COOLING_DOWN;

        E_METIS_CRYO_CTRL_CMD.WARM_UP:
            logs.M_LogInfo('Warm-Up initiated by operator from PARTIALLY_COLD state');
            stat.nState := E_METIS_CRYO_CTRL_STATE.WARMING_UP;

        ELSE
            logs.M_LogInfo('Unhandled command in PARTIALLY_COLD state');
            // Stay in current state
    END_CASE

ELSE
    // Keep Stabalization ON if no action is given
    M_Activity_Stabilize_Cryostat_Conditions();

END_IF

M_SetStatus(stat.nState);
RETURN;



//ctrl.bSafe_Evac 			:= TRUE;
//ctrl.bSafe_Cool_Down 		:= TRUE;
//ctrl.bSafe_Warm_Up 			:= TRUE;
//ctrl.bSafe_Regeneration 	:= FALSE;
//ctrl.bSafe_Anti_Fogging		:= TRUE;
//ctrl.bSafe_Venting 			:= FALSE;
//ctrl.bEnable_Venting		:= FALSE;
//stat.bPermitEvacuationStop 	:= FALSE;

//IF	ctrl.bExecute	THEN
//	ctrl.bExecute		:= FALSE;
//	stat.nLastCommand	:= ctrl.nCommand;
//	ctrl.nCommand		:= E_METIS_CRYO_CTRL_CMD.NONE;
//	IF stat.nLastCommand = E_METIS_CRYO_CTRL_CMD.COOL	THEN	
//		logs.M_LogInfo('Cool-Down initiated by operator');
//		stat.nState	:= E_METIS_CRYO_CTRL_STATE.COOLING_DOWN;
//	ELSIF stat.nLastCommand = E_METIS_CRYO_CTRL_CMD.WARM_UP	THEN
//		logs.M_LogInfo('Warm-Up initiated by operator');
//		stat.nState	:= E_METIS_CRYO_CTRL_STATE.WARMING_UP;
//	END_IF
//ELSE
//	M_Activity_Stabilize_Cryostat_Conditions();
//	stat.nState	:= E_METIS_CRYO_CTRL_STATE.PARTIALLY_COLD;
//END_IF

//M_SetStatus(stat.nState);	
//RETURN;
END_METHOD

METHOD M_Activity_Stabilize_Cryostat_Conditions : BOOL
VAR_INPUT
END_VAR




IF NOT stat.bEvacuationActive THEN
	ctrl.bSafe_Evac := TRUE;
	met_evac.M_Start_Evacuation();
END_IF

IF NOT stat.bWarm AND (stat.bInGoodVacuum OR stat.bInVacuum) THEN

	ctrl.bSafe_Anti_Fogging := TRUE;
	met_anti_fogging.M_Start_AntiFogging();
END_IF
END_METHOD

METHOD M_Activity_Venting : BOOL
VAR_INPUT
END_VAR

ctrl.bSafe_Cool_Down     := FALSE;
ctrl.bSafe_Warm_Up       := FALSE;
ctrl.bSafe_Evac          := FALSE;
ctrl.bSafe_Regeneration  := FALSE;
ctrl.bSafe_Venting 		 := TRUE;

// Stop Atomatic Evacuation

stat.sState := 'State: VENTING in progress...';

// Case 1: Venting completed successfully
IF stat.bVentingFinishedSuccessfully THEN
	ctrl.bEnable_Venting := FALSE;
	logs.M_LogInfo('VENTING completed successfully.');
	stat.nState := E_METIS_CRYO_CTRL_STATE.WARM_PRESS;
	stat.sState := 'State: Warm & Pressurized (Post-Vent)';
	logs.M_LogInfo('Transition to WARM_PRESS.');
	M_SetStatus(stat.nState);
	RETURN;
END_IF

// Case 2: Venting interrupted manually
IF trgVentingOff.Q THEN
	ctrl.bEnable_Venting := FALSE;
	logs.M_LogInfo('VENTING interrupted by operator.');

	IF stat.bPressurized THEN
		stat.nState := E_METIS_CRYO_CTRL_STATE.WARM_PRESS;
		stat.sState := 'State: Warm & Pressurized (Vent Interrupted)';
		logs.M_LogInfo('Fallback: WARM_PRESS.');
		
	ELSIF stat.bPartialVacuum THEN
		stat.nState := E_METIS_CRYO_CTRL_STATE.PARTIAL_VACUUM;
		stat.sState := 'State: Partial Vacuum (Vent Interrupted)';
		logs.M_LogInfo('Fallback: PARTIAL_VACUUM.');

	ELSIF stat.bInVacuum OR stat.bInGoodVacuum THEN
		stat.nState := E_METIS_CRYO_CTRL_STATE.WARM_VACUUM;
		stat.sState := 'State: Warm Vacuum (Vent Interrupted)';
		logs.M_LogInfo('Fallback: WARM_VACUUM.');
		
	ELSE
		stat.nState := E_METIS_CRYO_CTRL_STATE.ERROR;
		stat.sState := 'State: ERROR – Undefined pressure condition after venting abort.';
		//logs.M_LogError('Venting interrupted but system pressure condition undefined. Transitioning to ERROR.');
	END_IF

	M_SetStatus(stat.nState);
	RETURN;
END_IF


M_SetStatus(stat.nState);
RETURN;
END_METHOD

METHOD M_Activity_Warm_Press_State : BOOL
VAR_INPUT
END_VAR
	ctrl.bSafe_Evac 		:= TRUE;
	ctrl.bSafe_Cool_Down 	:= FALSE;
	ctrl.bSafe_Warm_Up		:= FALSE;
	ctrl.bSafe_Regeneration := FALSE;
	ctrl.bSafe_Venting 		:= FALSE;
	ctrl.bEnable_Venting 	:= FALSE;


	IF	ctrl.bExecute	THEN
		ctrl.bExecute		:= FALSE;
		stat.nLastCommand	:= ctrl.nCommand;
		ctrl.nCommand		:= E_METIS_CRYO_CTRL_CMD.NONE;
		IF stat.nLastCommand = E_METIS_CRYO_CTRL_CMD.NONE THEN
			logs.M_LogInfo('Cryo Controller Disables by operator');
			stat.nState	:= E_METIS_CRYO_CTRL_STATE.NONE;
			ctrl.bEnable := FALSE;
			stat.bInitialized := FALSE;
		END_IF
	ELSIF stat.bPartialVacuum THEN
		// Evacuation is not part of the State Machine.
		// Once the pressure is below ambient , we switch to Partial Vacuum.
		stat.nState := E_METIS_CRYO_CTRL_STATE.PARTIAL_VACUUM;
		logs.M_LogInfo('Transitioning to Partial Vacuum state: pressure < ambient.');
	END_IF
	
	M_SetStatus(stat.nState);	
	RETURN;
END_METHOD

METHOD M_Activity_Warm_Up_State : BOOL
VAR_INPUT
END_VAR
ctrl.bSafe_Evac            := TRUE;
ctrl.bSafe_Cool_Down       := FALSE;
ctrl.bSafe_Warm_Up         := TRUE;
ctrl.bSafe_Regeneration    := FALSE;
ctrl.bSafe_Venting         := FALSE;
ctrl.bEnable_Venting       := FALSE;
ctrl.bSafe_Anti_Fogging    := FALSE;

stat.bPermitEvacuationStop := FALSE;


// Wait for warm-up to complete or be aborted
IF trgWarmupOff.Q THEN
    ctrl.bEnable_Warm_Up := FALSE;

    IF stat.bWarm THEN
        logs.M_LogInfo('Warm-up complete. State is WARM_VACUUM');
        stat.nState := E_METIS_CRYO_CTRL_STATE.WARM_VACUUM;

    ELSIF stat.bPartiallyCold THEN
        logs.M_LogInfo('Warm-up complete. State is PARTIALLY_COLD');
        stat.nState := E_METIS_CRYO_CTRL_STATE.PARTIALLY_COLD;

    ELSIF stat.bOP THEN
        logs.M_LogWarning('Unexpected OP state detected after warm-up. Assuming COLD state');
        stat.nState := E_METIS_CRYO_CTRL_STATE.COLD;

    ELSE
        logs.M_LogWarning('Unknown thermal state after warm-up. Retaining current state.');
    END_IF
END_IF

M_SetStatus(stat.nState);
RETURN;
END_METHOD

METHOD M_Activity_Warm_Vacuum_State : BOOL
VAR_INPUT
END_VAR


IF stat.bRegenerationActive THEN
	ctrl.bSafe_Evac         := TRUE;
	ctrl.bSafe_Venting      := FALSE;
	ctrl.bSafe_Cool_Down    := FALSE;
	ctrl.bSafe_Regeneration := TRUE;
	ctrl.bSafe_Warm_Up      := FALSE;
	ctrl.bSafe_Anti_Fogging := FALSE; 
ELSE
	ctrl.bSafe_Evac         := TRUE;
	ctrl.bSafe_Venting      := TRUE;
	ctrl.bSafe_Cool_Down    := TRUE;
	ctrl.bSafe_Regeneration := TRUE;
	ctrl.bSafe_Warm_Up      := FALSE;
	ctrl.bSafe_Anti_Fogging := TRUE;
END_IF


// Evaluate execution command
IF ctrl.bExecute THEN
	ctrl.bExecute      := FALSE;
	stat.nLastCommand  := ctrl.nCommand;
	ctrl.nCommand      := E_METIS_CRYO_CTRL_CMD.NONE;

	CASE stat.nLastCommand OF

		E_METIS_CRYO_CTRL_CMD.COOL:
			// Preconditions for cooling down
			IF stat.bInVacuum THEN
				logs.M_LogInfo('Cool-Down initiated by operator.');
				stat.nState := E_METIS_CRYO_CTRL_STATE.COOLING_DOWN;
			ELSE
				logs.M_LogWarning('Cannot start Cool-Down: Good vacuum not reached.');
			END_IF

		E_METIS_CRYO_CTRL_CMD.VENT:
			logs.M_LogInfo('Venting initiated by operator.');
			stat.nState := E_METIS_CRYO_CTRL_STATE.VENTING;

		E_METIS_CRYO_CTRL_CMD.NONE:
			// No action — intentional idle
		ELSE
			logs.M_LogWarning(CONCAT('Unexpected command in Warm Vacuum: ', TO_STRING(stat.nLastCommand)));
	END_CASE
END_IF

M_SetStatus(stat.nState);
RETURN;
END_METHOD

METHOD M_CheckDetectorsSafety : BOOL
VAR_INPUT
END_VAR
END_METHOD

METHOD M_CheckDetectorTempStability
VAR_INPUT
END_VAR
END_METHOD

METHOD M_CheckForCommands
VAR_INPUT
END_VAR
// Capture system Enable/Disable command

trgSystemEnable(CLK := ctrl.bEnable);
trgSystemDisable(CLK := ctrl.bEnable);
// Capture System Disable
IF trgSystemDisable.Q THEN
	ctrl.bExecute	:= TRUE;
	ctrl.nCommand	:= E_METIS_CRYO_CTRL_CMD.NONE;
END_IF


// Capture Cool Down command
trgCool(CLK := ctrl.bEnable_Cool_Down);
trgCoolOFF(CLK := stat.bCoolDownActive);
IF	ctrl.bEnable_Cool_Down AND (stat.nState = E_METIS_CRYO_CTRL_STATE.WARM_VACUUM OR stat.nState = E_METIS_CRYO_CTRL_STATE.PARTIALLY_COLD) THEN
	ctrl.bExecute	:= TRUE;
	ctrl.nCommand	:= E_METIS_CRYO_CTRL_CMD.COOL;
END_IF



// Capture Warmup command

trgWarmup(CLK := ctrl.bEnable_Warm_Up);
trgWarmupOff(CLK := stat.bWarmUpActive);
IF	trgWarmup.Q AND 
	(stat.nState = E_METIS_CRYO_CTRL_STATE.COOLING_DOWN OR stat.nState = E_METIS_CRYO_CTRL_STATE.COLD) THEN
	ctrl.bExecute	:= TRUE;
	ctrl.nCommand	:= E_METIS_CRYO_CTRL_CMD.WARM_UP;
END_IF


// Capture Venting command
trgVenting(CLK := ctrl.bEnable_Venting);
trgVentingOff(CLK := ctrl.bEnable_Venting);

IF	trgVenting.Q THEN 
	IF (stat.nState = E_METIS_CRYO_CTRL_STATE.WARM_VACUUM) OR 
	   (stat.nState = E_METIS_CRYO_CTRL_STATE.PARTIAL_VACUUM) THEN
		ctrl.bExecute	:= TRUE;
		ctrl.nCommand	:= E_METIS_CRYO_CTRL_CMD.VENT;
	END_IF
END_IF


// Capture Evacuation ON/OFF trigger
trgEvacOn(CLK := ctrl.bEnable_Evac);
trgEvacOff(CLK := ctrl.bEnable_Evac);
IF	trgEvacOn.Q AND NOT ctrl.bEnable_Venting THEN
	ctrl.bEnable_Evac	:= TRUE;
	ctrl.bSafe_Evac := TRUE;
	M_SysLog('Evacuation started.');
ELSIF trgEvacOff.Q THEN
	ctrl.bEnable_Evac	:= FALSE;
	M_SysLog('Evacuation stopped.');
END_IF

// Capture Regeneration command
trgRegeneration(CLK := ctrl.bEnable_Regeneration);
trgRegenerationOff(CLK := ctrl.bEnable_Regeneration);
IF	trgRegeneration.Q AND (stat.nState = E_METIS_CRYO_CTRL_STATE.WARM_VACUUM) THEN  
	ctrl.bSafe_Regeneration := TRUE;
	M_SysLog('Regeneration started...');
ELSIF trgRegenerationOff.Q THEN
	ctrl.bEnable_Regeneration	:= FALSE;
	M_SysLog('Regeneration stopped');
END_IF
END_METHOD

METHOD M_CheckForSensorErrors
VAR_INPUT
END_VAR
//////////////////////////////////////////////////
//// Check for errors by testing the 'Valid' flag.
//////////////////////////////////////////////////
//IF		NOT Pressure_Cryo.stat.bValid	THEN
//	stat.bError	:= TRUE;
//	stat.sState	:= 'Cryo Vacuum gauge problem';
//	stat.nState	:= E_CRYO_CTRL_STATE.ERROR;
//ELSIF	NOT Temp_Mirror.stat.bValid	THEN
//	stat.bError	:= TRUE;
//	stat.sState	:= 'Mirror Temperature sensor problem';
//	stat.nState	:= E_CRYO_CTRL_STATE.ERROR;
//ELSE
//	stat.bError	:= FALSE;
//	stat.sState	:= '';
//END_IF


/////////////////////////
//// Check for Interlocks
/////////////////////////

////
//// Evacuation and Repressurization are mutually exclusive.
////
//IF EvacSys.in_bEnable THEN
//	ctrl.bEnable_RepressSys	:= FALSE;
//ELSIF RepressValve.in_bEnable THEN
//	ctrl.bEnable_Evac	:= FALSE;
//END_IF

////
//// Disable control in failure state
////
//IF stat.bError THEN
//	ctrl.bEnable_Precool	:= FALSE;
//	ctrl.bEnable_Cool 		:= FALSE;
//	ctrl.bEnable_Warmup		:= FALSE;
//END_IF
END_METHOD

METHOD M_CheckLakeshoreCommand
VAR_INPUT
END_VAR
(* TODO

IF ctrl.bLS_UpdateSETP THEN
	// Reset trigger flag
	ctrl.bLS_UpdateSETP	:= FALSE;
	
	// Safety
	IF ctrl.lrLS_RAMP > 1.0 THEN
		ctrl.lrLS_RAMP	:= 1.0;
	ELSIF ctrl.lrLS_RAMP < 0.0 THEN
		ctrl.lrLS_RAMP	:= 0.0;
	END_IF
	
